(*=======================================================*)
	1:	(* Warte auf Kommando *)
		IF st_ecd_cmd.enu_cmd > NO_COMMAND THEN
			IF st_ecd_cmd.enu_cmd <= HALT_AXIS THEN
				(* Wichtige Kommandos werden mit Direktsprung ausgeführt, um Zykluszeit zu sparen *)
				IF st_ecd_cmd.enu_cmd = HALT_AXIS THEN
					fb_state_entry.i16_next_step := 120;
				ELSIF st_ecd_cmd.enu_cmd = STOP_AXIS THEN
					fb_state_entry.i16_next_step := 130;
				ELSE
					fb_state_entry.i16_next_step := 10;	(* Motionbefehle *)
				END_IF
			ELSE
				fb_state_entry.i16_next_step := 500;	(* Parameter für Achsen *)
			END_IF
		END_IF

(*=======================Motionbefehle================================*)
	10:	(* Power OFF NC-Achse *)
		fb_ton_cmd_timeout.IN := TRUE;
		IF st_ecd_cmd.enu_cmd = POWER_DISABLE THEN
			mc_power_axis.Enable := FALSE;
			fb_state_entry.i16_next_step := 11;
		ELSE
			fb_ton_cmd_timeout.IN := FALSE;
			fb_state_entry.i16_next_step := 20;
		END_IF
	11:
		CASE i16_achstyp OF
			LINEAR, RUND:
				IF NOT mc_power_axis.Status AND NOT st_masterachse.Status.Operational THEN
					fb_state_entry.i16_next_step := 999;
				ELSIF NOT mc_power_axis.Busy AND mc_power_axis.Error THEN
					err_id := mc_power_axis.ErrorID;
					st_ecd_cmd.meldungen.sm_power_disable := TRUE;
					fb_state_entry.i16_next_step := 1000;
				END_IF
			LINEAR_VIRTUELL, RUND_VIRTUELL:
				IF NOT mc_power_axis.Busy AND mc_power_axis.Error THEN
					err_id := mc_power_axis.ErrorID;
					st_ecd_cmd.meldungen.sm_power_disable := TRUE;
					fb_state_entry.i16_next_step := 1000;
				ELSE
					fb_state_entry.i16_next_step := 999;
				END_IF
			SERVOKLEMME7201:
				IF NOT mc_power_axis.Status AND NOT st_masterachse.Status.Operational THEN
					fb_state_entry.i16_next_step := 999;
				ELSIF NOT mc_power_axis.Busy AND mc_power_axis.Error THEN
					err_id := mc_power_axis.ErrorID;
					st_ecd_cmd.meldungen.sm_power_disable := TRUE;
					fb_state_entry.i16_next_step := 1000;
				END_IF
		END_CASE

(*=======================================================*)
	20:	(* Reset NC-Achse und Servokontroller*)
		IF	st_ecd_cmd.enu_cmd = RESET OR
			st_masterachse.Status.DriveDeviceError OR
			st_masterachse.Status.Error
			 THEN
			fb_state_entry.i16_next_step := 21;
		ELSE
			fb_state_entry.i16_next_step := 30;
		END_IF
	21:	(*  Reset AX5000 Fehler  *)
		CASE i16_achstyp OF
			LINEAR, RUND:
				IF NOT st_masterachse.Status.DriveDeviceError THEN
					fb_state_entry.i16_next_step := 24;
				ELSE
					fb_ton_cmd_timeout.IN := TRUE;
					fb_soe_reset.Execute := TRUE;
					IF fb_soe_reset.Busy THEN
						fb_state_entry.i16_next_step := 22;
					END_IF
				END_IF
			LINEAR_VIRTUELL, RUND_VIRTUELL, SERVOKLEMME7201:
				fb_state_entry.i16_next_step := 24;
		END_CASE
	22:
		IF NOT fb_soe_reset.Busy THEN
			IF  fb_soe_reset.Error THEN
				st_ecd_cmd.meldungen.sm_reset := TRUE;
				fb_state_entry.i16_next_step := 1000;
			ELSE
				fb_soe_reset.Execute := FALSE;
				fb_state_entry.i16_next_step := 23;
			END_IF
		END_IF
	23:
		IF NOT st_masterachse.Status.DriveDeviceError THEN
			fb_ton_cmd_timeout.IN := FALSE;
			fb_state_entry.i16_next_step := 24;
		END_IF
	24:	(* Reset NC-Achsfehler *)
		CASE i16_achstyp OF
			LINEAR, RUND, LINEAR_VIRTUELL, RUND_VIRTUELL:
				IF NOT st_masterachse.Status.Error THEN
					fb_state_entry.i16_next_step := 26;
				ELSE
					fb_ton_cmd_timeout.IN := TRUE;
					mc_reset_axis.Execute := TRUE;
					IF mc_reset_axis.Busy THEN
						fb_state_entry.i16_next_step := 25;
					END_IF
				END_IF
			SERVOKLEMME7201:
				IF NOT st_masterachse.Status.Error AND NOT st_masterachse.Status.DriveDeviceError THEN
					fb_state_entry.i16_next_step := 26;
				ELSE
					fb_ton_cmd_timeout.IN := TRUE;
					mc_reset_axis.Execute := TRUE;
					IF mc_reset_axis.Busy THEN
						fb_state_entry.i16_next_step := 25;
					END_IF
				END_IF
		END_CASE
	25:
		IF NOT st_masterachse.Status.Error THEN
			mc_reset_axis.Execute := FALSE;
			fb_ton_cmd_timeout.IN := FALSE;
			fb_state_entry.i16_next_step := 26;
		END_IF
	26:
		IF st_ecd_cmd.enu_cmd = RESET THEN
			fb_state_entry.i16_next_step := 999;
		ELSE
			fb_state_entry.i16_next_step := 30;
		END_IF

(*=======================================================*)
	30:	(* Power ON NC-Achse *)
		CASE i16_achstyp OF
			LINEAR, RUND:
				fb_ton_cmd_timeout.IN := TRUE;
				IF	(st_ecd_cmd.enu_cmd > POWER_DISABLE AND st_ecd_cmd.enu_cmd < HALT_AXIS)  AND
					(NOT st_masterachse.Status.Operational OR
					(st_ecd_cmd.enu_cmd = POWER_ENABLE AND NOT st_masterachse.Status.Operational))
					THEN
						fb_state_entry.i16_next_step := 31;
				ELSE
					fb_ton_cmd_timeout.IN := FALSE;
					fb_state_entry.i16_next_step := 40;
				END_IF
			LINEAR_VIRTUELL, RUND_VIRTUELL, SERVOKLEMME7201:
				IF	st_ecd_cmd.enu_cmd > POWER_DISABLE AND st_ecd_cmd.enu_cmd < HALT_AXIS AND
					NOT mc_power_axis.Status
					THEN
						fb_state_entry.i16_next_step := 31;
				ELSE
					fb_ton_cmd_timeout.IN := FALSE;
					fb_state_entry.i16_next_step := 40;
				END_IF
		END_CASE
	31:
		mc_power_axis.Enable_Positive := TRUE;
		mc_power_axis.Enable_Negative := TRUE;
		mc_power_axis.Enable := TRUE;
		IF mc_power_axis.Busy THEN
			fb_ton_vz.PT := t#1s;
			fb_ton_vz.IN := TRUE;
			fb_state_entry.i16_next_step := 32;
		END_IF
	32:
		IF mc_power_axis.Status AND st_masterachse.Status.Operational  THEN
			IF st_ecd_cmd.enu_cmd = POWER_ENABLE THEN
				fb_state_entry.i16_next_step := 999;
			ELSE
				fb_ton_cmd_timeout.IN := FALSE;
				fb_state_entry.i16_next_step := 40;
			END_IF
		ELSIF mc_power_axis.Error AND fb_ton_vz.Q THEN
			st_ecd_cmd.meldungen.sm_power_enable := TRUE;
			err_id := mc_power_axis.ErrorID;
			fb_state_entry.i16_next_step := 1000;
		END_IF
		IF st_ecd_cmd.enu_cmd = HALT_AXIS THEN
			fb_ton_cmd_timeout.IN := FALSE;
			fb_ton_vz.IN := FALSE;
			fb_state_entry.i16_next_step := 121;
		END_IF
		IF st_ecd_cmd.enu_cmd = STOP_AXIS THEN
			fb_ton_cmd_timeout.IN := FALSE;
			fb_ton_vz.IN := FALSE;
			fb_state_entry.i16_next_step := 131;
		END_IF

(*=======================================================*)
	40:	(* Abfrage Referenzieren und Ref-Art *)
		IF st_ecd_cmd.enu_cmd = HOME THEN
			IF b_refsensor_vorhanden THEN
				mc_referenzmodus := MC_DefaultHoming;
			ELSE
				mc_referenzmodus := MC_Direct;
			END_IF
			st_position.r_referenz := 0.0;
			fb_state_entry.i16_next_step := 41;
		ELSE
			fb_ton_cmd_timeout.IN := FALSE;
			fb_state_entry.i16_next_step := 50;
		END_IF
	41:	(* Start Homing *)
		mc_home_axis.Execute := TRUE;
		mc_home_axis.Options.ClearPositionLag := TRUE;
		IF mc_home_axis.Busy THEN
			fb_state_entry.i16_next_step := 42;
		END_IF
	42:
		IF mc_home_axis.Done THEN
			mc_home_axis.Execute := FALSE;
			fb_state_entry.i16_next_step := 999;
		END_IF
		IF NOT mc_home_axis.Busy AND mc_home_axis.Error THEN
			st_ecd_cmd.meldungen.sm_home := TRUE;
			err_id := mc_home_axis.ErrorID;
			fb_state_entry.i16_next_step := 1000;
		END_IF
		IF st_ecd_cmd.enu_cmd = HALT_AXIS THEN
			mc_home_axis.Execute := FALSE;
			fb_ton_cmd_timeout.IN := FALSE;
			fb_state_entry.i16_next_step := 121;
		END_IF
		IF st_ecd_cmd.enu_cmd = STOP_AXIS THEN
			mc_home_axis.Execute := FALSE;
			fb_ton_cmd_timeout.IN := FALSE;
			fb_state_entry.i16_next_step := 131;
		END_IF

(*=======================================================*)
	50:	(* Jog vorwärts *)
		IF st_ecd_cmd.enu_cmd = JOG_VORWAERTS THEN
			fb_state_entry.i16_next_step := 51;
		ELSE
			fb_state_entry.i16_next_step := 55;
		END_IF
	51:
		b_jog_vorwaerts_execute := TRUE;
		IF mc_jog_axis.Active THEN
			fb_state_entry.i16_next_step := 52;
		ELSIF mc_jog_axis.Error THEN
			st_ecd_cmd.meldungen.sm_jog_vorwaerts := TRUE;
			fb_state_entry.i16_next_step := FEHLER;
		END_IF
	52:
		IF st_ecd_cmd.enu_cmd = JOG_STOP OR st_ecd_cmd.enu_cmd = JOG_RUECKWAERTS THEN
			fb_state_entry.i16_next_step := 61;
		END_IF

		IF st_ecd_cmd.enu_cmd = HALT_AXIS THEN
			mc_movemodulo_axis.Execute := FALSE;
			fb_ton_cmd_timeout.IN := FALSE;
			fb_state_entry.i16_next_step := 121;
		END_IF
		IF st_ecd_cmd.enu_cmd = STOP_AXIS THEN
			mc_movemodulo_axis.Execute := FALSE;
			fb_ton_cmd_timeout.IN := FALSE;
			fb_state_entry.i16_next_step := 131;
		END_IF

(*=======================================================*)
	55:	(* Jog rückwärts *)
		IF st_ecd_cmd.enu_cmd = JOG_RUECKWAERTS THEN
			fb_state_entry.i16_next_step := 56;
		ELSE
			fb_state_entry.i16_next_step := 60;
		END_IF

	56:
		b_jog_rueckwaerts_execute := TRUE;
		IF mc_jog_axis.Active THEN
			fb_state_entry.i16_next_step := 57;
		ELSIF mc_jog_axis.Error THEN
			st_ecd_cmd.meldungen.sm_jog_rueckwaerts := TRUE;
			fb_state_entry.i16_next_step := FEHLER;
		END_IF
	57:
		IF st_ecd_cmd.enu_cmd = JOG_STOP OR st_ecd_cmd.enu_cmd = JOG_VORWAERTS THEN
			fb_state_entry.i16_next_step := 61;
		END_IF

		IF st_ecd_cmd.enu_cmd = HALT_AXIS THEN
			mc_movemodulo_axis.Execute := FALSE;
			fb_ton_cmd_timeout.IN := FALSE;
			fb_state_entry.i16_next_step := 121;
		END_IF
		IF st_ecd_cmd.enu_cmd = STOP_AXIS THEN
			mc_movemodulo_axis.Execute := FALSE;
			fb_ton_cmd_timeout.IN := FALSE;
			fb_state_entry.i16_next_step := 131;
		END_IF

(*=======================================================*)
	60:	(* Jog Stop *)
		IF st_ecd_cmd.enu_cmd = JOG_STOP THEN
			fb_state_entry.i16_next_step := 61;
		ELSE
			fb_state_entry.i16_next_step := 70;
		END_IF
	61:
		b_jog_vorwaerts_execute := FALSE;
		b_jog_rueckwaerts_execute := FALSE;
		fb_state_entry.i16_next_step := 999;

(*=======================================================*)
	70:	(* Move absolute *)
		IF st_ecd_cmd.enu_cmd = MOVE_ABSOLUTE THEN
			fb_state_entry.i16_next_step := 71;
		ELSE
			fb_state_entry.i16_next_step := 80;
		END_IF
	71:
		IF ABS(st_masterachse.NcToPlc.ActPos -  st_position.r_soll ) < 0.05 THEN
			fb_state_entry.i16_next_step := 999;
		ELSE
			mc_moveabsolute_axis.Execute := TRUE;
		END_IF
		IF mc_moveabsolute_axis.Busy THEN
			fb_state_entry.i16_next_step := 72;
		END_IF
	72:
		IF mc_moveabsolute_axis.Done THEN
			mc_moveabsolute_axis.Execute := FALSE;
			fb_state_entry.i16_next_step := 999;
		END_IF
		IF NOT mc_moveabsolute_axis.Busy AND mc_moveabsolute_axis.Error THEN
			st_ecd_cmd.meldungen.sm_move_absolute := TRUE;
			err_id := mc_moveabsolute_axis.ErrorID;
			fb_state_entry.i16_next_step := 1000;
		END_IF
		IF st_ecd_cmd.enu_cmd = HALT_AXIS THEN
			mc_moveabsolute_axis.Execute := FALSE;
			fb_ton_cmd_timeout.IN := FALSE;
			fb_state_entry.i16_next_step := 121;
		END_IF
		IF st_ecd_cmd.enu_cmd = STOP_AXIS THEN
			mc_moveabsolute_axis.Execute := FALSE;
			fb_ton_cmd_timeout.IN := FALSE;
			fb_state_entry.i16_next_step := 131;
		END_IF

		(* Move-Kommando für folgende Bewegung *)
		IF st_ecd_cmd.enu_cmd = MOVE_ABSOLUTE_NEXT THEN
			fb_state_entry.i16_next_step := 74;
		END_IF
	74:
		IF ABS(st_masterachse.NcToPlc.ActPos -  st_position.r_soll ) < 0.05 THEN
			fb_state_entry.i16_next_step := 999;
		ELSE
			mc_moveabsolutenext_axis.Execute := TRUE;
		END_IF
		IF mc_moveabsolutenext_axis.Busy THEN
			fb_state_entry.i16_next_step := 75;
		END_IF
	75:
		IF mc_moveabsolutenext_axis.Done THEN
			mc_moveabsolute_axis.Execute := FALSE;
			mc_moveabsolutenext_axis.Execute := FALSE;
			fb_state_entry.i16_next_step := 999;
		END_IF
		IF NOT mc_moveabsolutenext_axis.Busy AND mc_moveabsolutenext_axis.Error THEN
			st_ecd_cmd.meldungen.sm_move_absolute := TRUE;
			err_id := mc_moveabsolutenext_axis.ErrorID;
			fb_state_entry.i16_next_step := 1000;
		END_IF
		IF st_ecd_cmd.enu_cmd = HALT_AXIS THEN
			mc_moveabsolute_axis.Execute := FALSE;
			mc_moveabsolutenext_axis.Execute := FALSE;
			fb_ton_cmd_timeout.IN := FALSE;
			fb_state_entry.i16_next_step := 121;
		END_IF
		IF st_ecd_cmd.enu_cmd = STOP_AXIS THEN
			mc_moveabsolute_axis.Execute := FALSE;
			mc_moveabsolutenext_axis.Execute := FALSE;
			fb_ton_cmd_timeout.IN := FALSE;
			fb_state_entry.i16_next_step := 131;
		END_IF

(*=======================================================*)
	80:	(* Move relative *)
		IF st_ecd_cmd.enu_cmd = MOVE_RELATIVE THEN
			fb_state_entry.i16_next_step := 81;
		ELSE
			fb_state_entry.i16_next_step := 90;
		END_IF
	81:
		mc_moverelative_axis.Execute := TRUE;
		IF mc_moverelative_axis.Busy THEN
			fb_state_entry.i16_next_step := 82;
		END_IF
	82:
		IF mc_moverelative_axis.Done THEN
			mc_moverelative_axis.Execute := FALSE;
			fb_state_entry.i16_next_step := 999;
		END_IF
		IF NOT mc_moverelative_axis.Busy AND mc_moverelative_axis.Error THEN
			st_ecd_cmd.meldungen.sm_move_relative := TRUE;
			err_id := mc_moverelative_axis.ErrorID;
			fb_state_entry.i16_next_step := 1000;
		END_IF
		IF st_ecd_cmd.enu_cmd = HALT_AXIS THEN
			mc_moverelative_axis.Execute := FALSE;
			fb_ton_cmd_timeout.IN := FALSE;
			fb_state_entry.i16_next_step := 121;
		END_IF
		IF st_ecd_cmd.enu_cmd = STOP_AXIS THEN
			mc_moverelative_axis.Execute := FALSE;
			fb_ton_cmd_timeout.IN := FALSE;
			fb_state_entry.i16_next_step := 131;
		END_IF

(*=======================================================*)
	90:	(* Move velocity *)
		IF st_ecd_cmd.enu_cmd = MOVE_VELOCITY THEN
			fb_state_entry.i16_next_step := 91;
		ELSE
			fb_state_entry.i16_next_step := 100;
		END_IF
	91:
		mc_movevelocity_axis.Execute := TRUE;
		IF mc_movevelocity_axis.Busy THEN
			fb_state_entry.i16_next_step := 92;
		END_IF
	92:
		IF mc_movevelocity_axis.InVelocity THEN
			mc_movevelocity_axis.Execute := FALSE;
			fb_state_entry.i16_next_step := 999;
		END_IF
		IF NOT mc_movevelocity_axis.Busy AND mc_movevelocity_axis.Error THEN
			st_ecd_cmd.meldungen.sm_move_velocity := TRUE;
			err_id := mc_movevelocity_axis.ErrorID;
			fb_state_entry.i16_next_step := 1000;
		END_IF
		IF st_ecd_cmd.enu_cmd = HALT_AXIS THEN
			mc_movevelocity_axis.Execute := FALSE;
			fb_ton_cmd_timeout.IN := FALSE;
			fb_state_entry.i16_next_step := 121;
		END_IF
		IF st_ecd_cmd.enu_cmd = STOP_AXIS THEN
			mc_movevelocity_axis.Execute := FALSE;
			fb_ton_cmd_timeout.IN := FALSE;
			fb_state_entry.i16_next_step := 131;
		END_IF

(*=======================================================*)
	100:	(* Move modulo *)
		IF st_ecd_cmd.enu_cmd = MOVE_MODULO THEN
			fb_state_entry.i16_next_step := 101;
		ELSE
			fb_state_entry.i16_next_step := 103;
		END_IF
	101:
		IF ABS(st_masterachse.NcToPlc.ModuloActPos -  st_position.r_soll ) < 0.3 THEN
			fb_state_entry.i16_next_step := 999;
		ELSE
			mc_movemodulo_axis.Execute := TRUE;
		END_IF
		IF mc_movemodulo_axis.Busy THEN
			fb_state_entry.i16_next_step := 102;
		END_IF
	102:
		IF mc_movemodulo_axis.Done THEN
			mc_movemodulo_axis.Execute := FALSE;
			fb_state_entry.i16_next_step := 999;
		END_IF

		IF NOT mc_movemodulo_axis.Busy AND mc_movemodulo_axis.Error THEN
			st_ecd_cmd.meldungen.sm_move_modulo := TRUE;
			err_id := mc_movemodulo_axis.ErrorID;
			fb_state_entry.i16_next_step := 1000;
		END_IF
		IF st_ecd_cmd.enu_cmd = HALT_AXIS THEN
			mc_movemodulo_axis.Execute := FALSE;
			fb_ton_cmd_timeout.IN := FALSE;
			fb_state_entry.i16_next_step := 121;
		END_IF
		IF st_ecd_cmd.enu_cmd = STOP_AXIS THEN
			mc_movemodulo_axis.Execute := FALSE;
			fb_ton_cmd_timeout.IN := FALSE;
			fb_state_entry.i16_next_step := 131;
		END_IF

(*=======================================================*)
	103:
		(*Touch Probe checken*)
		IF	fb_state_entry.E THEN
			mc_abort_trigger.Execute:=TRUE;
		END_IF

		IF st_ecd_cmd.enu_cmd = MOVE_TOUCH_PROBE THEN

			(*Touch Probe darf nicht betätigt sein*)
			IF	(b_FallingEdge AND NOT b_TriggerInput) OR
				(NOT b_FallingEdge AND b_TriggerInput)  THEN
				st_ecd_cmd.meldungen.sm_touch_probe_defect := TRUE;		(*Messtaster defekt*)
				fb_state_entry.i16_next_step := FEHLER;

			ELSIF mc_abort_trigger.Done THEN
				lr_RecPos:=0;
				fb_state_entry.i16_next_step := 104;
			END_IF

		ELSE
			fb_state_entry.i16_next_step := 110;
		END_IF

		IF	fb_state_entry.X THEN
			mc_abort_trigger.Execute:=FALSE;
		END_IF

	104:
		(* Move absolute (Position muss hinter dem Touch Probe liegen => der Restweg wird gelöscht)*)
		IF 	ABS(st_masterachse.NcToPlc.ActPos -  st_position.r_soll ) < 0.05 THEN
			fb_state_entry.i16_next_step := 999;
		ELSE
			mc_moveabsolute_axis.Execute := TRUE;
			mc_touch_probe.Execute:=TRUE;
		END_IF
		IF 	mc_moveabsolute_axis.Busy THEN
			fb_state_entry.i16_next_step := 105;
		END_IF

	105:
		(*Achsposition wurde erreicht ohne Taster Event*)
		IF 	mc_moveabsolute_axis.Done THEN
			fb_state_entry.i16_next_step := 999;
		END_IF

		(*Achse anhalten wenn Touch Probe betätigt wird*)
		IF 	mc_moveabsolute_axis.Busy AND
			(b_TriggerInput = NOT b_FallingEdge OR
			mc_touch_probe.Done) THEN
			fb_state_entry.i16_next_step := 131;
		END_IF

		(*Übergabe Rec Position*)
		IF	mc_touch_probe.Done THEN
			lr_RecPos:=mc_touch_probe.RecordedPosition;
		END_IF

		(*Fehler Achse*)
		IF 	NOT mc_moveabsolute_axis.Busy AND mc_moveabsolute_axis.Error THEN
			st_ecd_cmd.meldungen.sm_move_absolute := TRUE;
			err_id := mc_moveabsolute_axis.ErrorID;
			fb_state_entry.i16_next_step := FEHLER;
		END_IF

		(*Fehler Touch Probe*)
		IF  	mc_touch_probe.Error THEN
			st_ecd_cmd.meldungen.sm_touch_probe_err := TRUE;
			err_id := mc_touch_probe.ErrorID;
			fb_state_entry.i16_next_step := FEHLER;
		END_IF

		IF	fb_state_entry.X THEN
			fb_ton_cmd_timeout.IN := FALSE;
			mc_moveabsolute_axis.Execute := FALSE;
			mc_touch_probe.Execute:=FALSE;
		END_IF

(*=======================================================*)
	110:	(* Position *)
		IF st_ecd_cmd.enu_cmd = SET_POSITION THEN
			fb_state_entry.i16_next_step := 111;
		ELSE
			fb_state_entry.i16_next_step := 121;
		END_IF
	111:
		(* Soll- und Istposition werden auf den gleichen Wert gesetzt und somit der Schleppfehler gelöscht. *)
		mc_setposition_axis.Options.ClearPositionLag := TRUE;
		mc_setposition_axis.Options.EncoderIndex := 0;
		mc_setposition_axis.Options.SelectEncoderIndex := FALSE;
		mc_setposition_axis.Execute := TRUE;
		IF mc_setposition_axis.Busy THEN
			fb_state_entry.i16_next_step := 112;
		END_IF
	112:
		IF mc_setposition_axis.Done THEN
			mc_setposition_axis.Execute := FALSE;
			fb_state_entry.i16_next_step := 999;
		END_IF
		IF NOT mc_setposition_axis.Busy AND mc_setposition_axis.Error THEN
			st_ecd_cmd.meldungen.sm_setposition := TRUE;
			err_id := mc_setposition_axis.ErrorID;
			fb_state_entry.i16_next_step := 1000;
		END_IF
		IF st_ecd_cmd.enu_cmd = HALT_AXIS THEN
			mc_setposition_axis.Execute := FALSE;
			fb_ton_cmd_timeout.IN := FALSE;
			fb_state_entry.i16_next_step := 121;
		END_IF
		IF st_ecd_cmd.enu_cmd = STOP_AXIS THEN
			mc_setposition_axis.Execute := FALSE;
			fb_ton_cmd_timeout.IN := FALSE;
			fb_state_entry.i16_next_step := 131;
		END_IF

(*=======================================================*)
	120:	(* Halt *)
		fb_ton_cmd_timeout.IN := TRUE;
		IF st_ecd_cmd.enu_cmd = HALT_AXIS THEN
			fb_state_entry.i16_next_step := 121;
		ELSE
			fb_ton_cmd_timeout.IN := FALSE;
			fb_state_entry.i16_next_step := 131;
		END_IF
	121:
		mc_halt_axis.Execute := TRUE;
		IF mc_halt_axis.Busy THEN
			fb_state_entry.i16_next_step := 122;
		END_IF
	122:
		IF mc_halt_axis.Done THEN
			mc_halt_axis.Execute := FALSE;
			fb_state_entry.i16_next_step := 123;
		END_IF
		IF NOT mc_halt_axis.Busy AND mc_halt_axis.Error THEN
			st_ecd_cmd.meldungen.sm_halt_axis := TRUE;
			err_id := mc_halt_axis.ErrorID;
			fb_state_entry.i16_next_step := 1000;
		END_IF
	123:
		IF	NOT st_masterachse.Status.ConstantVelocity AND
			NOT st_masterachse.Status.Accelerating AND
			NOT st_masterachse.Status.Decelerating
			THEN
				fb_state_entry.i16_next_step := 999;
		END_IF

(*=======================================================*)
	130: (* Stop *)
		fb_ton_cmd_timeout.IN := TRUE;
		IF st_ecd_cmd.enu_cmd = STOP_AXIS THEN
			fb_state_entry.i16_next_step := 131;
		ELSE
			fb_ton_cmd_timeout.IN := FALSE;
			fb_state_entry.i16_next_step := 140;
		END_IF
	131:
		mc_stop_axis.Execute := TRUE;
		IF mc_stop_axis.Busy THEN
			fb_state_entry.i16_next_step := 132;
		END_IF
	132:
		IF mc_stop_axis.Done THEN
			mc_stop_axis.Execute := FALSE;
			fb_state_entry.i16_next_step := 133;
		END_IF
		IF mc_stop_axis.Error THEN
			st_ecd_cmd.meldungen.sm_stop_axis := TRUE;
			err_id := mc_stop_axis.ErrorID;
			fb_state_entry.i16_next_step := 1000;
		END_IF
	133:
		IF 	NOT st_masterachse.Status.ConstantVelocity AND
			NOT st_masterachse.Status.Accelerating AND
			NOT st_masterachse.Status.Decelerating
			THEN
				fb_state_entry.i16_next_step := 999;
		END_IF

(*=======================================================*)
	140:	(* Frei *)
		fb_state_entry.i16_next_step := 500;

(*======================Parameterbefehle=================================*)
	500:	(* Schreibe einen Parameter an den Antrieb *)
		fb_ton_cmd_timeout.IN := TRUE;
		IF st_ecd_cmd.enu_cmd = SOE_WRITE_PARAM THEN
			fb_state_entry.i16_next_step := 501;
		ELSE
			fb_ton_cmd_timeout.IN := FALSE;
			fb_state_entry.i16_next_step := 510;
		END_IF
	501:
		fb_soe_write.Execute := TRUE;
		IF fb_soe_write.Busy THEN
			fb_state_entry.i16_next_step := 502;
		END_IF
	502:
		IF NOT fb_soe_write.Busy THEN
			fb_soe_write.Execute := FALSE;
			IF fb_soe_write.Error THEN
				st_ecd_cmd.meldungen.sm_write_soe_parameter := TRUE;
				fb_state_entry.i16_next_step := 1000;
			ELSE
				fb_state_entry.i16_next_step := 999;
			END_IF
		END_IF

(*=======================================================*)
	510:	(* Lesen eines Parameter vom Antrieb *)
		fb_ton_cmd_timeout.IN := TRUE;
		IF st_ecd_cmd.enu_cmd = SOE_READ_PARAM THEN
			fb_state_entry.i16_next_step := 511;
		ELSE
			fb_ton_cmd_timeout.IN := FALSE;
			fb_state_entry.i16_next_step := 520;
		END_IF
	511:
		fb_soe_read.Execute := TRUE;
		IF fb_soe_read.Busy THEN
			fb_state_entry.i16_next_step := 512;
		END_IF
	512:
		IF NOT fb_soe_read.Busy THEN
			fb_soe_write.Execute := FALSE;
			IF fb_soe_read.Error THEN
				st_ecd_cmd.meldungen.sm_read_soe_parameter := TRUE;
				fb_state_entry.i16_next_step := 1000;
			ELSE
				fb_state_entry.i16_next_step := 999;
			END_IF
		END_IF

(*=======================================================*)
	520:	(* Schreibe einen Parameter an die NC-Achse *)
		fb_ton_cmd_timeout.IN := TRUE;
		IF st_ecd_cmd.enu_cmd = WRITE_NC_PARAMETER THEN
			fb_state_entry.i16_next_step := 521;
		ELSE
			fb_ton_cmd_timeout.IN := FALSE;
			fb_state_entry.i16_next_step := 530;
		END_IF
	521:
		mc_write_nc_parameter.Execute := TRUE;
		IF mc_write_nc_parameter.Busy THEN
			fb_state_entry.i16_next_step := 522;
		END_IF
	522:
		IF NOT mc_write_nc_parameter.Busy THEN
			mc_write_nc_parameter.Execute := FALSE;
			IF mc_write_nc_parameter.Error THEN
				st_ecd_cmd.meldungen.sm_write_nc_parameter := TRUE;
				fb_state_entry.i16_next_step := 1000;
			ELSE
				fb_state_entry.i16_next_step := 999;
			END_IF
		END_IF

(*=======================================================*)
	530:	(* Lesen eines Parameter vom der NC-Achse *)
		fb_ton_cmd_timeout.IN := TRUE;
		IF st_ecd_cmd.enu_cmd = READ_NC_PARAMETER THEN
			fb_state_entry.i16_next_step := 531;
		ELSE
			fb_ton_cmd_timeout.IN := FALSE;
			fb_state_entry.i16_next_step := 540;
		END_IF
	531:
		mc_read_nc_parameter.Enable := TRUE;
		IF mc_read_nc_parameter.Busy THEN
			fb_state_entry.i16_next_step := 532;
		END_IF
	532:
		IF NOT mc_read_nc_parameter.Busy THEN
			mc_read_nc_parameter.Enable := FALSE;
			IF mc_read_nc_parameter.Error THEN
				st_ecd_cmd.meldungen.sm_read_nc_parameter := TRUE;
				fb_state_entry.i16_next_step := 1000;
			ELSE
				fb_state_entry.i16_next_step := 999;
			END_IF
		END_IF

(*=======================================================*)
	540:	(* Schreibe einen beliebigen ADS-Parameter an die NC-Achse *)
		fb_ton_cmd_timeout.IN := TRUE;
		IF st_ecd_cmd.enu_cmd = WRITE_ADS_PARAMETER THEN
			fb_state_entry.i16_next_step := 541;
		ELSE
			fb_ton_cmd_timeout.IN := FALSE;
			fb_state_entry.i16_next_step := 550;
		END_IF
	541:
		fb_ads_write.WRITE := TRUE;
		IF fb_ads_write.BUSY THEN
			fb_state_entry.i16_next_step := 542;
		END_IF
	542:
		IF NOT fb_ads_write.BUSY THEN
			fb_ads_write.WRITE := FALSE;
			IF fb_ads_write.ERR THEN
				st_ecd_cmd.meldungen.sm_write_ads_parameter := TRUE;
				fb_state_entry.i16_next_step := 1000;
			ELSE
				fb_state_entry.i16_next_step := 999;
			END_IF
		END_IF

(*=======================================================*)
	550:	(* Lesen einen beliebigenADS-Parameter vom der NC-Achse *)
		fb_ton_cmd_timeout.IN := TRUE;
		IF st_ecd_cmd.enu_cmd = READ_ADS_PARAMETER THEN
			fb_state_entry.i16_next_step := 551;
		ELSE
			fb_ton_cmd_timeout.IN := FALSE;
			fb_state_entry.i16_next_step := 560;
		END_IF
	551:
		fb_ads_read.READ := TRUE;
		IF fb_ads_read.BUSY THEN
			fb_state_entry.i16_next_step := 552;
		END_IF
	552:
		IF NOT fb_ads_read.BUSY THEN
			fb_ads_read.READ := FALSE;
			IF fb_ads_read.ERR THEN
				st_ecd_cmd.meldungen.sm_read_ads_parameter := TRUE;
				fb_state_entry.i16_next_step := 1000;
			ELSE
				fb_state_entry.i16_next_step := 999;
			END_IF
		END_IF

(*=======================================================*)
	560:	(* Schreibe die neuen EcSoe Parameter an den Antrieb *)
		fb_ton_cmd_timeout.IN := TRUE;
		IF st_ecd_cmd.enu_cmd = ECCOESDO_WRITE_PARAM THEN
			fb_state_entry.i16_next_step := 561;
		ELSE
			fb_ton_cmd_timeout.IN := FALSE;
			fb_state_entry.i16_next_step := 570;
		END_IF
	561:
		fb_ec_coe_sdo_write_ex.bExecute := TRUE;
		IF fb_ec_coe_sdo_write_ex.bBusy THEN
			fb_state_entry.i16_next_step := 562;
		END_IF
	562:
		IF NOT fb_ec_coe_sdo_write_ex.bBusy THEN
			fb_ec_coe_sdo_write_ex.bExecute := FALSE;
			IF fb_ec_coe_sdo_write_ex.bError THEN
				st_ecd_cmd.meldungen.sm_ec_coe_sdo_write_ex := TRUE;
				fb_state_entry.i16_next_step := 1000;
			ELSE
				fb_state_entry.i16_next_step := 999;
			END_IF
		END_IF

(*=======================================================*)
	570:	(* Lese die neuen EcSoe Parameter an den Antrieb *)
		fb_ton_cmd_timeout.IN := TRUE;
		IF st_ecd_cmd.enu_cmd = ECCOESDO_READ_PARAM THEN
			fb_state_entry.i16_next_step := 571;
		ELSE
			fb_ton_cmd_timeout.IN := FALSE;
			fb_state_entry.i16_next_step := 580;
		END_IF
	571:
		fb_ec_coe_sdo_read_ex.bExecute := TRUE;
		IF fb_ec_coe_sdo_read_ex.bBusy THEN
			fb_state_entry.i16_next_step := 572;
		END_IF
	572:
		IF NOT fb_ec_coe_sdo_read_ex.bBusy THEN
			fb_ec_coe_sdo_read_ex.bExecute := FALSE;
			IF fb_ec_coe_sdo_read_ex.bError THEN
				st_ecd_cmd.meldungen.sm_ec_coe_sdo_read_ex := TRUE;
				fb_state_entry.i16_next_step := 1000;
			ELSE
				fb_state_entry.i16_next_step := 999;
			END_IF
		END_IF

(*=======================================================*)
	580:	(* Frei *)
		fb_state_entry.i16_next_step := 999;

(*=======================================================*)
	999:	(* Ende - Befehl wurde korrekt abgearbeitet *)
		st_ecd_cmd.enu_cmd := NO_COMMAND;
		fb_ton_cmd_timeout.IN := FALSE;
		fb_ton_vz.IN := FALSE;

		b_jog_vorwaerts_execute := FALSE;
		b_jog_rueckwaerts_execute := FALSE;

		mc_reset_axis.Execute := FALSE;
		mc_home_axis.Execute := FALSE;
		mc_moveabsolute_axis.Execute := FALSE;
		mc_moverelative_axis.Execute := FALSE;
		mc_movevelocity_axis.Execute := FALSE;
		mc_movemodulo_axis.Execute := FALSE;
		mc_setposition_axis.Execute := FALSE;
		mc_halt_axis.Execute := FALSE;
		mc_stop_axis.Execute := FALSE;
		fb_soe_reset.Execute := FALSE;
		fb_soe_write.Execute := FALSE;
		fb_soe_read.Execute := FALSE;
		mc_write_nc_parameter.Execute := FALSE;
		mc_read_nc_parameter.Enable := FALSE;
		fb_ads_write.WRITE := FALSE;
		fb_ads_read.READ := FALSE;
		fb_ec_coe_sdo_write_ex.bExecute := FALSE;
		fb_ec_coe_sdo_read_ex.bExecute := FALSE;

		st_ecd_cmd.meldungen.sm_power_enable := FALSE;
		st_ecd_cmd.meldungen.sm_power_disable := FALSE;
		st_ecd_cmd.meldungen.sm_reset := FALSE;
		st_ecd_cmd.meldungen.sm_home := FALSE;
		st_ecd_cmd.meldungen.sm_setposition := FALSE;
		st_ecd_cmd.meldungen.sm_jog_vorwaerts := FALSE;
		st_ecd_cmd.meldungen.sm_jog_rueckwaerts := FALSE;
		st_ecd_cmd.meldungen.sm_move_absolute := FALSE;
		st_ecd_cmd.meldungen.sm_move_relative := FALSE;
		st_ecd_cmd.meldungen.sm_move_velocity := FALSE;
		st_ecd_cmd.meldungen.sm_move_modulo := FALSE;
		st_ecd_cmd.meldungen.sm_stop_axis := FALSE;
		st_ecd_cmd.meldungen.sm_halt_axis := FALSE;
		st_ecd_cmd.meldungen.sm_motion_command_timeout := FALSE;
		st_ecd_cmd.meldungen.sm_limit_positiv_erreicht := FALSE;
		st_ecd_cmd.meldungen.sm_limit_negativ_erreicht := FALSE;
		st_ecd_cmd.meldungen.sm_write_soe_parameter := FALSE;
		st_ecd_cmd.meldungen.sm_read_soe_parameter := FALSE;
		st_ecd_cmd.meldungen.sm_write_nc_parameter := FALSE;
		st_ecd_cmd.meldungen.sm_read_nc_parameter := FALSE;
		st_ecd_cmd.meldungen.sm_write_ads_parameter := FALSE;
		st_ecd_cmd.meldungen.sm_read_ads_parameter := FALSE;
		st_ecd_cmd.meldungen.sm_ec_coe_sdo_write_ex := FALSE;
		st_ecd_cmd.meldungen.sm_ec_coe_sdo_read_ex := FALSE;

		fb_state_entry.i16_next_step := 1;

(*=======================================================*)
	1000: (* Fehler *)
		IF fb_state_entry.E THEN
			st_ecd_cmd.b_job_fehler := TRUE;
			fb_ton_cmd_timeout.IN := FALSE;
			fb_ton_vz.IN := FALSE;
			st_ecd_cmd.enu_cmd := NO_COMMAND;
		END_IF

		(* Fehler reseten *)
		IF st_ecd_cmd.enu_cmd >= ABORT THEN
			st_ecd_cmd.b_job_fehler := FALSE;
			b_jog_vorwaerts_execute := FALSE;
			b_jog_rueckwaerts_execute := FALSE;
			mc_reset_axis.Execute := FALSE;
			mc_home_axis.Execute := FALSE;
			mc_moveabsolute_axis.Execute := FALSE;
			mc_moverelative_axis.Execute := FALSE;
			mc_movevelocity_axis.Execute := FALSE;
			mc_movemodulo_axis.Execute := FALSE;
			mc_setposition_axis.Execute := FALSE;
			mc_halt_axis.Execute := FALSE;
			mc_stop_axis.Execute := FALSE;
			fb_soe_reset.Execute := FALSE;
			fb_soe_write.Execute := FALSE;
			fb_soe_read.Execute := FALSE;
			mc_write_nc_parameter.Execute := FALSE;
			mc_read_nc_parameter.Enable := FALSE;
			fb_ads_write.WRITE := FALSE;
			fb_ads_read.READ := FALSE;
			fb_ec_coe_sdo_write_ex.bExecute := FALSE;
			fb_ec_coe_sdo_read_ex.bExecute := FALSE;
			fb_state_entry.i16_next_step := 0;
		END_IF
END_CASE

(* Endlagenüberwachung der maximalen Verfahrwege der Achse *)
IF b_limitsensor_positiv_vorhanden AND fb_f_trig_limit_sensor_positiv.Q THEN
	mc_stop_axis.Execute := TRUE;
	st_ecd_cmd.meldungen.sm_limit_positiv_erreicht := TRUE;
	fb_state_entry.i16_next_step := 1000;
END_IF
IF b_limitsensor_negativ_vorhanden AND fb_f_trig_limit_sensor_negativ.Q THEN
	mc_stop_axis.Execute := TRUE;
	st_ecd_cmd.meldungen.sm_limit_negativ_erreicht := TRUE;
	fb_state_entry.i16_next_step := 1000;
END_IF

(* Timeout-Fehler aller Drivekommandos *)
IF fb_ton_cmd_timeout.Q THEN
	fb_ton_cmd_timeout.IN := FALSE;
	st_ecd_cmd.meldungen.sm_motion_command_timeout := TRUE;
	fb_state_entry.i16_next_step := 1000;
END_IF

(*Abbruch des aktuellen Achskommandos *)
IF st_ecd_cmd.enu_cmd = ABORT AND fb_state_entry.i16_next_step <> FEHLER THEN
	fb_state_entry.i16_next_step := 999;
END_IF

(* Statehistory *)
fb_state_entry(
	i16_next_step:= ,
	i16_pos:= 2,
	s_debugtext:= ,
	E=> , 
	X=> , 
	i16_step=> ,
	i16_last_step=> );

fb_cmd_history(i16_current_cmd:= st_ecd_cmd.enu_cmd, last_cmd=> );

(*=============================================================================================*)
(* Ab hier werden alle Verfahraufträge für eine Achse abgewickelt *)

(* Lese Zustand der Achse *)
st_masterachse.ReadStatus;

(* Für Rundachsen muss die Sollgeschwindigkeit umgerechnet werden in °/s *)
IF i16_achstyp = RUND OR i16_achstyp = RUND_VIRTUELL THEN
	lr_sollgeschwindigkeit := lr_sollgeschwindigkeit * 360 / 60;
END_IF

(*=============================================================================================*)
(* Reglerfreigabe *)
mc_power_axis(
	Enable:= ,
	Enable_Positive:= ,
	Enable_Negative:= ,
	Override:= lr_override,
	BufferMode:= mc_buffermode_axis,
	Axis:= st_masterachse,
	Status=> ,
	Busy=> ,
	Active=> ,
	Error=> ,
	ErrorID=> );

(*=============================================================================================*)
(* Achse aus Fehlerzustand rücksetzen *)
(* NC-Achse *)
mc_reset_axis(
	Execute:= ,
	Axis:= st_masterachse,
	Done=> ,
	Busy=> ,
	Error=> ,
	ErrorID=> );

(* AX5000 Servokontroller *)
fb_soe_reset(
	NetId:= , 
	Execute:= , 
	Timeout:= t_ads_timeout,
	Axis:= st_masterachse,
	Busy=> ,
	Error=> , 
	AdsErrId=> , 
	SercosErrId=> );

(*=============================================================================================*)
(* Achsposition setzen *)
mc_setposition_axis(
	Execute:= ,
	Position:= st_position.r_soll,
	Mode:= FALSE, (* RELATIVE=True, ABSOLUTE=False (Default) *)
	Options:= ,
	Axis:= st_masterachse,
	Done=> ,
	Busy=> ,
	Error=> ,
	ErrorID=> );

(*=============================================================================================*)
(* Achse referenzieren *)
mc_home_axis(
	Execute:= ,
	Position:= st_position.r_referenz,
	HomingMode:= mc_referenzmodus,
	BufferMode:= mc_buffermode_axis,
	Options:= ,
	bCalibrationCam:= e_referenznocken,
	Axis:= st_masterachse,
	Done=> ,
	Busy=> ,
	Active=> ,
	CommandAborted=> ,
	Error=> ,
	ErrorId=> );

(*=============================================================================================*)
(* Achse tippen *)
mc_jog_axis(
	JogForward:= b_jog_vorwaerts_execute AND NOT b_jog_rueckwaerts_execute,
	JogBackwards:= b_jog_rueckwaerts_execute AND NOT b_jog_vorwaerts_execute,
	Mode:= MC_JOGMODE_CONTINOUS,  (* motion with standard jog parameters for slow motion *)
	Velocity:= lr_sollgeschwindigkeit,
	Acceleration:= st_vorgabe_geschwindigkeiten.lr_beschleunigung,
	Deceleration:= st_vorgabe_geschwindigkeiten.lr_verzoegerung,
	Jerk:= st_vorgabe_geschwindigkeiten.lr_ruck,
	Axis:= st_masterachse,
	Done=> ,
	Busy=> ,
	Active=> ,
	CommandAborted=> ,
	Error=> ,
	ErrorId=> );

(*=============================================================================================*)
(* Fahre Achse absolut *)
mc_moveabsolute_axis(
	Execute:= ,
	Position:= st_position.r_soll,
	Velocity:= lr_sollgeschwindigkeit,
	Acceleration:= st_vorgabe_geschwindigkeiten.lr_beschleunigung,
	Deceleration:= st_vorgabe_geschwindigkeiten.lr_verzoegerung,
	Jerk:= st_vorgabe_geschwindigkeiten.lr_ruck,
	BufferMode:= mc_buffermode_axis,
	Options:= ,
	Axis:= st_masterachse,
	Done=> ,
	Busy=> ,
	Active=> ,
	CommandAborted=> ,
	Error=> ,
	ErrorID=> );
(* Fahre Achse absolut im Falle einer Folgebewegung *)
mc_moveabsolutenext_axis(
	Execute:= ,
	Position:= st_position.r_soll,
	Velocity:= lr_sollgeschwindigkeit,
	Acceleration:= st_vorgabe_geschwindigkeiten.lr_beschleunigung,
	Deceleration:= st_vorgabe_geschwindigkeiten.lr_verzoegerung,
	Jerk:= st_vorgabe_geschwindigkeiten.lr_ruck,
	BufferMode:= mc_buffermode_axis,
	Options:= ,
	Axis:= st_masterachse,
	Done=> ,
	Busy=> ,
	Active=> ,
	CommandAborted=> ,
	Error=> ,
	ErrorID=> );

(*=============================================================================================*)
(* Fahre Achse relaiv *)
mc_moverelative_axis(
	Execute:= ,
	Distance:= st_position.r_soll,
	Velocity:= lr_sollgeschwindigkeit,
	Acceleration:= st_vorgabe_geschwindigkeiten.lr_beschleunigung,
	Deceleration:= st_vorgabe_geschwindigkeiten.lr_verzoegerung,
	Jerk:= st_vorgabe_geschwindigkeiten.lr_ruck,
	BufferMode:= mc_buffermode_axis,
	Options:= ,
	Axis:= st_masterachse,
	Done=> ,
	Busy=> ,
	Active=> ,
	CommandAborted=> ,
	Error=> ,
	ErrorID=> );

(*=============================================================================================*)
(* Gleichlaufachse starten *)
mc_movevelocity_axis(
	Execute:= ,
	Velocity:= lr_sollgeschwindigkeit,
	Acceleration:= st_vorgabe_geschwindigkeiten.lr_beschleunigung,
	Deceleration:= st_vorgabe_geschwindigkeiten.lr_verzoegerung,
	Jerk:= st_vorgabe_geschwindigkeiten.lr_ruck,
	Direction:= mc_richtung_velocity,
	BufferMode:= mc_buffermode_axis,
	Options:= ,
	Axis:= st_masterachse,
	InVelocity=> ,
	Busy=> ,
	Active=> ,
	CommandAborted=> ,
	Error=> ,
	ErrorID=> );

(*=============================================================================================*)
(* Bewegen einer Rundachse *)
mc_movemodulo_axis(
	Execute:= ,
	Position:= st_position.r_soll,
	Velocity:= lr_sollgeschwindigkeit,
	Acceleration:= st_vorgabe_geschwindigkeiten.lr_beschleunigung,
	Deceleration:= st_vorgabe_geschwindigkeiten.lr_verzoegerung,
	Jerk:= st_vorgabe_geschwindigkeiten.lr_ruck,
	Direction:= mc_richtung_modulo,
	BufferMode:= mc_buffermode_axis,
	Options:= ,
	Axis:= st_masterachse,
	Done=> ,
	Busy=> ,
	Active=> ,
	CommandAborted=> ,
	Error=> ,
	ErrorID=> );

(*=============================================================================================*)
mc_stop_axis(
	Execute:= ,
	Deceleration:= st_vorgabe_geschwindigkeiten.lr_verzoegerung,
	Jerk:= st_vorgabe_geschwindigkeiten.lr_ruck,
	Options:= ,
	Axis:= st_masterachse,
	Done=> ,
	Busy=> ,
	Active=> ,
	CommandAborted=> ,
	Error=> ,
	ErrorID=> );

(*=============================================================================================*)
(* MC_Halt führt einen normalen Halt während der Bewegung aus.
Im Gegensatz dazu verriegelt MC_Stop die Achse gegen weitere Bewegungskommandos und
sollte nur in besonderen Situationen angewendet werden. *)
mc_halt_axis(
	Execute:= ,
	Deceleration:= st_vorgabe_geschwindigkeiten.lr_verzoegerung,
	Jerk:= st_vorgabe_geschwindigkeiten.lr_ruck,
	BufferMode:= mc_buffermode_axis,
	Options:= ,
	Axis:= st_masterachse,
	Done=> ,
	Busy=> ,
	Active=> ,
	CommandAborted=> ,
	Error=> ,
	ErrorID=> );

(*=============================================================================================*)
(* Einen Parameter auf den Antrieb schreiben *)
fb_soe_write(
	NetId:= , 
	Idn:= w_idn,	(* Idn := S_0_IDN + 33; *)
	Element:= EC_SOE_ELEMENT_VALUE,
	pSrcBuf:= ADR(ui16_soeparam_write_value),
	BufLen:= SIZEOF(ui16_soeparam_write_value),
	Execute:= , 
	Timeout:= t_ads_timeout,
	Password:= ,
	Axis:= st_masterachse,
	Busy=> ,
	Error=> ,
	AdsErrId=> ,
	SercosErrId=> );

(*=============================================================================================*)
(* Einen Parameter auf dem Antrieb lesen  *)
fb_soe_read(
	NetId:= , 
	Idn:= w_idn,	(* Idn := S_0_IDN + 33; *)
	Element:= EC_SOE_ELEMENT_VALUE,
	pDstBuf:= ADR(ui16_soeparam_read_value),
	BufLen:= SIZEOF(ui16_soeparam_read_value),
	Execute:= , 
	Timeout:= t_ads_timeout,
	Axis:= st_masterachse,
	Busy=> ,
	Error=> , 
	AdsErrId=> ,
	SercosErrId=> , 
	Attribute=> );

(*=============================================================================================*)
(* Einen Parameter auf die NC-Achse schreiben *)
mc_write_nc_parameter(
	Execute:= , 
	ParameterNumber:= i16_nc_parameter_nummer,
	Value:= r_wert_nc_write_parameter,
	Axis:= st_masterachse,
	Done=> ,
	Busy=> ,
	Error=> , 
	ErrorID=> );

(*=============================================================================================*)
(* Einen Parameter von der NC-Achse lesen *)
mc_read_nc_parameter(
	Enable:= , 
	ParameterNumber:= i16_nc_parameter_nummer,
	ReadMode:= READMODE_ONCE,
	Axis:= st_masterachse,
	Valid=> ,
	Busy=> ,
	Error=> , 
	ErrorID=> , 
	Value=> r_wert_nc_read_parameter);

(*=============================================================================================*)
(* Einen beliebigen ADS-Parameter auf die NC-Achse schreiben *)
fb_ads_write(
	NETID:= ,
	PORT:= 501,
	IDXGRP:= st_ads_info.st_symbol_info.idxGroup,
	IDXOFFS:= st_ads_info.st_symbol_info.idxOffset,
	LEN:= st_ads_info.st_symbol_info.byteSize,
	SRCADDR:= st_ads_info.dw_quelladresse_ads_write,
	WRITE:= ,
	TMOUT:= t_ads_timeout,
	BUSY=> , 
	ERR=> , 
	ERRID=> );

(*=============================================================================================*)
(* Einen beliebigen ADS-Parameter von der NC-Achse lesen *)
fb_ads_read(
	NETID:= ,
	PORT:= 501,
	IDXGRP:= st_ads_info.st_symbol_info.idxGroup,
	IDXOFFS:= st_ads_info.st_symbol_info.idxOffset,
	LEN:= st_ads_info.st_symbol_info.byteSize,
	DESTADDR:= st_ads_info.dw_zieladresse_ads_read,
	READ:= , 
	TMOUT:= t_ads_timeout,
	BUSY=> , 
	ERR=> , 
	ERRID=> );

(*=============================================================================================*)
(* Einen neuen EcCoeSdo-Parameter auf den Antrieb schreiben *)
fb_ec_coe_sdo_write_ex(
	sNetId:= st_eccoe_sdo.s_ec_slave_net_id,
	nSlaveAddr:= st_eccoe_sdo.ui16_slave_addr,
	nSubIndex:= st_eccoe_sdo.i8_sub_index,
	nIndex:= st_eccoe_sdo.w_index,
	pSrcBuf:= st_eccoe_sdo.dw_p_source_buffer,
	cbBufLen:= st_eccoe_sdo.ui32_buffer_length,
	bExecute:= ,
	tTimeout:= t_ads_timeout,
	bCompleteAccess:= FALSE,
	bBusy=> , 
	bError=> ,
	nErrId=> );

(*=============================================================================================*)
(* Einen neuen EcCoeSdo-Parameter von dem Antrieb lesen *)
fb_ec_coe_sdo_read_ex(
	sNetId:= st_eccoe_sdo.s_ec_slave_net_id,
	nSlaveAddr:= st_eccoe_sdo.ui16_slave_addr,
	nSubIndex:= st_eccoe_sdo.i8_sub_index,
	nIndex:= st_eccoe_sdo.w_index,
	pDstBuf:= st_eccoe_sdo.dw_p_destination_buffer,
	cbBufLen:= st_eccoe_sdo.ui32_buffer_length,
	bExecute:= ,
	tTimeout:= t_ads_timeout,
	bCompleteAccess:= FALSE,
	bBusy=> ,
	bError=> ,
	nErrId=> );
END_FUNCTION_BLOCK
ACTION sub_TouchProbe:
(*======================================================
   Command: MOVE_TOUCH_PROBE
 ------------------------------------------------------
   Auth: 		Werner Friedl    						 
   Date: 		10.09.2019    						     
   Rev.: 		1.0	
   Desc:		Mit diesem Command kann die Achsposition zu eimem Tastzeitpunkt aufgezeichnet werden.

			- im Achsaufruf müssen diese Einstellungen gemacht werden
		z.B.		b_TriggerInput:=i16_DigitalInput.0		=> Verknüpfung mit den Prozessdaten der Achse an dem der Taster angeklemmt wurde				
				i16_TouchProbeInNo:=1					=> 1 wenn der Taster am Input 1 angeklemmt wurde
				b_SignalEdge:=FallingEdge				=> FallingEdge ODER RisingEdge

		- das Kommando MOVE_TOUCH_PROBE fährt die Achse auf den Taster. Wird der Taster 
			während der Fahrt betätigt , dann stoppt die Achse automatisch und 
			das Messergebniss landet in der VAR lr_RecPos
		
		- Schritt103 => Taster prüfen
		- Schritt104 => Move Absolut und start Touch Probe
		- Schritt105 => Stop Achse und Übergabe Recording Position an die VAR lr_RecPos


		Konfiguration:
		In der IE Hilfe unter "Funktion Probe Unit" findet man die Beschreibung.
		
		im tsm muss der Touch Probe konfiguriert werden.
		Parameter		Wert		
		S-0-0303		405
		S-0-0307		409
		S-0-0169		1
		S-0-0170		3

		in den Prozessdaten einfügen 
		S-0-0801		Digital inputs, sate			und mit der Var i16_DigitalInput der jeweiligen Achse verknüpfen

		im Drivemanager die Logik der Probe unit einstellen 
		- bei Mux1 den Input auswählen und negiert zuweisen
		- 1: Auto activation from SafeOp to Op auswählen

		PLC:
		im VAR_OUTPUT der Achse die Var anlegen
		lr_RecPos							: LREAL;
		
		im VAR anlegen
		i16_DigitalInput						AT %I* : INT;
	
	
		und im Aufruf fb_axis die Var hinzufügen
	
		lr_RecPos=> lr_RecPos,
		b_TriggerInput:=i16_DigitalInput.2,
		b_FallingEdge:=TRUE


 ========================================================*)
IF	mc_touch_probe.Done THEN
	lr_RecPos:=mc_touch_probe.RecordedPosition;
END_IF


(* Touch Probe Initialisierung *)
TriggerInput.EncoderID:= 	st_masterachse.NcToPlc.AxisId;		(* funktioniert so nur wenn die Encoder ID gleich ist wie die Achs ID*)
TriggerInput.TouchProbe:=	TouchProbe1;					(*bei MC_TouchProbe immer TouchProbe1*)
TriggerInput.Edge:=			RisingEdge;						(*bei MC_TouchProbe immer RisingEdge*)
TriggerInput.Mode:=			TOUCHPROBEMODE_SINGLE;



(* Touch Probe Aufruf *)
mc_touch_probe(
	Execute:= ,
	WindowOnly:= 	FALSE ,
	FirstPosition:= ,
	LastPosition:= ,
	Axis:= 			st_masterachse,
	TriggerInput:=	TriggerInput ,
	Done=> ,
	Busy=> ,
	CommandAborted=> ,
	Error=> ,
	ErrorID=> ,
	RecordedPosition=> );

mc_abort_trigger(
	Execute:= ,
	Axis:= 			st_masterachse,
	TriggerInput:=	TriggerInput ,
	Done=> ,
	Busy=> ,
	Error=> , 
	ErrorID=> );
END_ACTION

(* POU EPT Lib/Funktionsbausteine/ST_CommandHistory, ST *)
FUNCTION_BLOCK ST_CommandHistory
VAR_INPUT
	i16_current_cmd 		: enum_ecd_cmd;
END_VAR
VAR_OUTPUT
	last_cmd 			: enum_ecd_cmd;
END_VAR
VAR
	arr_last_cmd_history 	: ARRAY[0..31] OF enum_ecd_cmd;
	i					: INT;
END_VAR
IF (last_cmd <> i16_current_cmd) THEN
	last_cmd := i16_current_cmd;

	FOR i:= 30 TO 0 BY -1DO
		arr_last_cmd_history[i+1] := arr_last_cmd_history[i];
	END_FOR
	arr_last_cmd_history[0] := last_cmd;
END_IF
END_FUNCTION_BLOCK

(* POU EPT Lib/Funktionsbausteine/ST_OT_UT_Ueberwachung, ST *)
FUNCTION_BLOCK ST_OT_UT_Ueberwachung
VAR_INPUT
	lr_achsposition				 : LREAL;
END_VAR
VAR_OUTPUT
	b_error						: BOOL;
END_VAR
VAR
	i32_anfang_ot					: DINT := 0;
	i32_ende_ot					: DINT := 5;
	i32_anfang_ut					: DINT := 180;
	i32_ende_ut					: DINT := 185;
	arr_eintrag					: ARRAY[0..99] OF BOOL := 1,0,1;	(* Länge dient nur zum Nachverfolgen *)
	b_ot							: BOOL := FALSE;
	b_ut							: BOOL := FALSE;
	fb_r_trig_ot					: R_TRIG;
	fb_r_trig_ut					: R_TRIG;
	fb_f_trig_ot					: F_TRIG;
	fb_f_trig_ut					: F_TRIG;
	i							: INT := 0;
END_VAR
(* Kontrollfunktion zum Prüfen, ob auf OT auch immer UT kommt. *)
(* Die Fehlerausgabe erfolgt mittels temporärer Fehlermeldung, welche im Errorlog der Visu mitgeschrieben wird. *)
(* Dies dient der Kontrolle auf fehlbedienung durch das Anlagenpersonal. *)

(* Flanken *)
fb_r_trig_ot(CLK:= b_ot, Q=> );
fb_r_trig_ut(CLK:= b_ut, Q=> );
fb_f_trig_ot(CLK:= b_ot, Q=> );
fb_f_trig_ut(CLK:= b_ut, Q=> );

(* Erstellen der Bereichsnocken *)
IF LREAL_TO_DINT(lr_achsposition) > i32_anfang_ot AND LREAL_TO_DINT(lr_achsposition) < i32_ende_ot THEN
	b_ot := TRUE;
	b_error := FALSE;
ELSE
	b_ot := FALSE;
END_IF

IF LREAL_TO_DINT(lr_achsposition) > i32_anfang_ut AND LREAL_TO_DINT(lr_achsposition) < i32_ende_ut THEN
	b_ut := TRUE;
	b_error := FALSE;
ELSE
	b_ut := FALSE;
END_IF

(* Eintragen von OT bzw. UT in das Register *)
IF fb_r_trig_ot.Q THEN
	FOR i := 99  TO 1 BY -1 DO
		arr_eintrag [i] := arr_eintrag[i - 1];
	END_FOR
	arr_eintrag[0] := 2#0;	(* Eintrag für OT = 0 *)
END_IF

IF fb_r_trig_ut.Q THEN
	FOR i := 99  TO 1 BY -1 DO
		arr_eintrag[i] := arr_eintrag[i - 1];
	END_FOR
	arr_eintrag[0] := 2#1;	(* Eintrag für UT = 1 *)
END_IF

(* Auswertung und Fehler *)
IF fb_f_trig_ot.Q OR fb_f_trig_ut.Q THEN
	b_error := NOT (arr_eintrag[0]  XOR arr_eintrag[1]);
END_IF
END_FUNCTION_BLOCK

(* POU Gemeinsamkeiten17xx/Bedienen/ST_Euchner_Handbedienpult, ST *)
PROGRAM ST_Euchner_Handbedienpult
VAR
	(* Eingänge von der Hardware *)
	e_Taste_Zustimm			AT %I* : BOOL;
	e_Taste_Plus				AT %I* : BOOL;
	e_Taste_Power			AT %I* : BOOL;
	e_Taste_Minus			AT %I* : BOOL;

	e_i16_Zaehler			AT %I* : INT;

	(* Instanzen *)
	fb_ton					: TON;

	(* Merker *)
	i16_merkpos				: INT := 0;
END_VAR
VAR_OUTPUT
	b_Taste_Zustimm			: BOOL := FALSE;
	b_Taste_Plus				: BOOL := FALSE;
	b_Taste_Power			: BOOL := FALSE;
	b_Taste_Minus			: BOOL := FALSE;

	i16_Handrad_delta		: INT := 0;
END_VAR
(* Tasten *)
b_Taste_Zustimm	:= e_Taste_Zustimm;
b_Taste_Plus	:= e_Taste_Plus;
b_Taste_Power := e_Taste_Power;
b_Taste_Minus := e_Taste_Minus;

(* Generiere Impuls für Delta Zähler *)
fb_ton(IN:= NOT fb_ton.Q , PT:= t#100ms, Q=> , ET=> );

IF fb_ton.Q THEN
	i16_Handrad_delta := e_i16_Zaehler - i16_merkpos;
	i16_merkpos := e_i16_Zaehler;
END_IF
END_PROGRAM

(* POU Gemeinsamkeiten17xx/Bedienen/ST_TippTasten, ST *)
PROGRAM ST_TippTasten
VAR_INPUT
	(* Geschwindigkeit / Stufe *)
	i16_akt_stufe						: INT := 0;	(* 0-9 *)
	b_initialisierungsphase				: BOOL := FALSE;
	b_einfaedeln_aktiv				: BOOL := FALSE;
END_VAR
VAR_IN_OUT
	st_visu							: struct_visu;
	st_visu_hinten						: struct_visu_hinten;
END_VAR
VAR
	lr_override						: LREAL := 25;
	lr_override_gestuft					: LREAL := 10;
	r_trig_tippen						: R_TRIG;
	r_trig_tippen_einfaedeln			: R_TRIG;
	r_trig_vorgabe					: R_TRIG;
	b_freigabe_override_auto			: BOOL := FALSE;
	fb_r_trig_quittieren					: R_TRIG;
END_VAR

VAR CONSTANT
	lr_override_init_einfaedel			: LREAL := 25;
END_VAR
(* Mit den zeitlichen Impulsen vom Handrad lässt sich der Override aller Achsen verändern. Die Geschwindigkeit wird im "ST_AxisJobCtrl_Motion" limitiert. *)
(* Tipp-Taste *)

r_trig_tippen(
		CLK:=NOT b_einfaedeln_aktiv AND (st_visu.b_tippen_start OR visu_hinten.out.b_start OR ST_Euchner_Handbedienpult.b_Taste_Power),
		Q=> );
r_trig_tippen_einfaedeln(
		CLK:= b_einfaedeln_aktiv AND (st_visu_hinten.out.b_tippen OR ST_Euchner_Handbedienpult.b_Taste_Power),
		Q=> );
r_trig_vorgabe(
		CLK:= st_visu.b_geschwindigkeit_vorgabe, Q=> );

(* Flanken *)
fb_r_trig_quittieren(CLK:= st_visu.b_quittieren OR st_visu_hinten.out.b_quittieren, Q=> );

CASE gi16_betriebsart OF
	AUTO:
		gb_ba_auto_kontroller := TRUE;

		IF r_trig_tippen.Q OR fb_r_trig_quittieren.Q THEN
			b_freigabe_override_auto := TRUE;
		END_IF

		IF b_einfaedeln_aktiv OR b_initialisierungsphase THEN
			lr_override := lr_override_gestuft := lr_override_init_einfaedel;
		ELSE

			IF r_trig_vorgabe.Q THEN
				i16_akt_stufe := 9;
			END_IF
			IF b_freigabe_override_auto THEN
				(* Override für Achsen mit "Vollgas" im Automatikbetrieb *)
				lr_override := 100;
				(* Override für Achsen, welche in Abstufung gefahren werden *)
				IF  i16_akt_stufe>= 0 AND i16_akt_stufe<= 9 THEN
					(* Overridevorgabe im Automatikbetrieb *)
					lr_override_gestuft := (i16_akt_stufe +1) * 10;
				ELSE
					(* Falls Geschwindigkeitsstufe was anderes als 0-9 enthält: Override auf 0: Keine Achse fährt *)
					lr_override_gestuft := 0;
				END_IF
			ELSE
				lr_override := lr_override_gestuft := 0;
			END_IF
		END_IF

	TIPPEN:
		b_freigabe_override_auto := FALSE;

		IF r_trig_tippen.Q OR lr_override > 0 OR  lr_override_gestuft > 0 THEN
			gb_ba_auto_kontroller := TRUE;
		ELSE
			gb_ba_auto_kontroller := FALSE;
		END_IF

		IF ST_Euchner_Handbedienpult.i16_Handrad_delta > 0 THEN
			lr_override := lr_override_gestuft := ABS(ST_Euchner_Handbedienpult.i16_Handrad_delta) * 0.1;
		ELSE
			lr_override := lr_override_gestuft := 0;
		END_IF

	HAND:
		gb_ba_auto_kontroller := FALSE;
		b_freigabe_override_auto := FALSE;
		lr_override := lr_override_gestuft := ABS(ST_Euchner_Handbedienpult.i16_Handrad_delta)* 0.1;
END_CASE

(* Abfrage maximaler Override grösser 100% *)
IF lr_override > 100 THEN
	lr_override := 100;
END_IF
IF lr_override_gestuft > 100 THEN
	lr_override_gestuft := 100;
END_IF
END_PROGRAM

(* POU Gemeinsamkeiten17xx/Achsen/ST_MotionFunctionPoints, ST *)
PROGRAM ST_MotionFunctionPoints
VAR_INPUT
	st_ctrl_in								: struct_ctrl_in;
END_VAR
VAR_OUTPUT
	st_ctrl_out							: struct_ctrl_out;
END_VAR
VAR
	fb_ton_wz							: TON;
	fb_ton_quitt							: TON;
	fb_state_entry						: ST_StateEntry;
	i, j									: INT := 0;
	udi_table_id_bestueckachse			: UDINT := 0;
	arr_motion_function_points		: ARRAY[1..ARRAY_LAENGE_MFP] OF struct_db_motionfunctionpoint;
END_VAR
VAR CONSTANT
	ARRAY_LAENGE_MFP				: INT := 100;
	YZTischMasterPos2					 : LREAL := 125;
	YZTischMasterPos3					 : LREAL := 185;
END_VAR
(* Zeiten *)
fb_ton_wz(IN:= ,PT:= , Q=>  , ET=> );
fb_ton_quitt(IN:= , PT:= t#50ms, Q=> , ET=> );

(* =====Berechnung MFPs===== *)
(* Berechnung von Punkten in einer Kurvenscheibe und der maximalen Mastergeschwindigkeit *)

(* =====Kopplung: Virtuelle Masterachse <-> Z-Achse ===== *)
fb_edit_mfps_bestuecken_z.fb(
	st_config:= fb_edit_mfps_bestuecken_z.st_config,
	st_ctrl_in:= fb_edit_mfps_bestuecken_z.st_ctrl.in,
	udiTableId:= 1,
	eMotionFunctionType:= MOTIONFUNCTYPE_POLYNOM5,
	i16_startpunkt_edit_mf_tab:= 2,
	arr_db_mf_tab:= arr_motion_function_points,
	lrVeloMax:= ST_Z_Achse.st_geschwindigkeiten.lr_maximalgeschwindigkeit,
	lrAccMax:= ST_Z_Achse.st_geschwindigkeiten.lr_beschleunigung,
	lrDecMax:= ST_Z_Achse.st_geschwindigkeiten.lr_verzoegerung,
	lrModuloValue:= 360.0,
	st_AxisRefMaster:= virtuelle_master_achse,
	st_AxisRefSlave:= z_achse,
	lrMasterVeloMax=> ,		(* Maximum Master Velocity [°/s] *)
	lrMasterRotPerMinMax=> ,	(* Maximum Master Rotations per Minute [1/min] *)
	st_ctrl_out=> fb_edit_mfps_bestuecken_z.st_ctrl.out);

(* =====Kopplung: Virtuelle Masterachse <-> Y-Achse ===== *)
fb_edit_mfps_bestuecken_y.fb(
	st_config:= fb_edit_mfps_bestuecken_y.st_config,
	st_ctrl_in:= fb_edit_mfps_bestuecken_y.st_ctrl.in,
	udiTableId:= 3,
	eMotionFunctionType:= MOTIONFUNCTYPE_POLYNOM5,
	i16_startpunkt_edit_mf_tab:= 2,
	arr_db_mf_tab:= arr_motion_function_points,
	lrVeloMax:= ST_Y_Achse.st_geschwindigkeiten.lr_maximalgeschwindigkeit,
	lrAccMax:= ST_Y_Achse.st_geschwindigkeiten.lr_beschleunigung,
	lrDecMax:= ST_Y_Achse.st_geschwindigkeiten.lr_verzoegerung,
	lrModuloValue:= 360.0,
	st_AxisRefMaster:= virtuelle_master_achse,
	st_AxisRefSlave:= y_achse,
	lrMasterVeloMax=> ,		(* Maximum Master Velocity [°/s] *)
	lrMasterRotPerMinMax=> ,	(* Maximum Master Rotations per Minute [1/min] *)
	st_ctrl_out=> fb_edit_mfps_bestuecken_y.st_ctrl.out);

(* =====Kopplung: Virtuelle Masterachse <-> Servobandeinzug-Achse ===== *)
fb_edit_mfps_bestuecken_b.fb(
	st_config:= fb_edit_mfps_bestuecken_b.st_config,
	st_ctrl_in:= fb_edit_mfps_bestuecken_b.st_ctrl.in,
	udiTableId:= 4,
	eMotionFunctionType:= MOTIONFUNCTYPE_POLYNOM5,
	i16_startpunkt_edit_mf_tab:= 2,
	arr_db_mf_tab:= arr_motion_function_points,
	lrVeloMax:= ST_Servobandeinzug.st_geschwindigkeiten.lr_maximalgeschwindigkeit,
	lrAccMax:= ST_Servobandeinzug.st_geschwindigkeiten.lr_beschleunigung,
	lrDecMax:= ST_Servobandeinzug.st_geschwindigkeiten.lr_verzoegerung,
	lrModuloValue:= 360.0,
	st_AxisRefMaster:= bestueckachse,
	st_AxisRefSlave:= b_achse,
	lrMasterVeloMax=> ,		(* Maximum Master Velocity [°/s] *)
	lrMasterRotPerMinMax=> ,	(* Maximum Master Rotations per Minute [1/min] *)
	st_ctrl_out=> fb_edit_mfps_bestuecken_b.st_ctrl.out);

(* =====Kopplung: Z-Achse <-> Y-Achse ===== *)
fb_edit_mfps_yz_tisch.fb(
	st_config:= fb_edit_mfps_yz_tisch.st_config,
	st_ctrl_in:= fb_edit_mfps_yz_tisch.st_ctrl.in,
	udiTableId:= 2,
	eMotionFunctionType:= MOTIONFUNCTYPE_POLYNOM5,
	i16_startpunkt_edit_mf_tab:= 2,
	arr_db_mf_tab:= arr_motion_function_points,
	lrVeloMax:= ST_Y_Achse.st_geschwindigkeiten.lr_maximalgeschwindigkeit,
	lrAccMax:= ST_Y_Achse.st_geschwindigkeiten.lr_beschleunigung,
	lrDecMax:= ST_Y_Achse.st_geschwindigkeiten.lr_verzoegerung,
	lrModuloValue:= 0.0,
	st_AxisRefMaster:= z_achse,
	st_AxisRefSlave:= y_achse,
	lrMasterVeloMax=> ,		(* Maximum Master Velocity [mm/s] *)
	lrMasterRotPerMinMax=> ,	(* Maximum Master Rotations per Minute [1/min] *)
	st_ctrl_out=> fb_edit_mfps_yz_tisch.st_ctrl.out);

(* =====Kopplung: Virtuelle Masterachse <-> Bestueckachse ===== *)
(*
fb_edit_mfps_bestueckachse.fb(
	st_config:= fb_edit_mfps_bestueckachse.st_config,
	st_ctrl_in:= fb_edit_mfps_bestueckachse.st_ctrl.in,
	udiTableId:= udi_table_id_bestueckachse,
	eMotionFunctionType:= MOTIONFUNCTYPE_POLYNOM5,
	i16_startpunkt_edit_mf_tab:= 1,
	arr_db_mf_tab:= gst_datensatz.st_wkz.st_virtmaster_bestueckachse.arr_motion_function_points,
	lrVeloMax:= ST_Bestueckachse.st_geschwindigkeiten.lr_maximalgeschwindigkeit,
	lrAccMax:= ST_Bestueckachse.st_geschwindigkeiten.lr_beschleunigung,
	lrDecMax:= ST_Bestueckachse.st_geschwindigkeiten.lr_verzoegerung,
	lrModuloValue:= 360.0,
	st_AxisRefMaster:= virtuelle_master_achse,
	st_AxisRefSlave:= bestueckachse,
	lrMasterVeloMax=> ,		(* Maximum Master Velocity [°/s] *)
	lrMasterRotPerMinMax=> ,	(* Maximum Master Rotations per Minute [1/min] *)
	st_ctrl_out=> fb_edit_mfps_bestueckachse.st_ctrl.out);
*)
fb_camtable_bestueckachse.fb(
	st_config:= fb_camtable_bestueckachse.st_config,
	st_ctrl_in:= fb_camtable_bestueckachse.st_ctrl.in,
	udiTableId:= udi_table_id_bestueckachse,
	arr_db_mf_tab:= arr_motion_function_points,
	lrModuloValue:= 360,
	st_AxisRefMaster:= virtuelle_master_achse,
	st_AxisRefSlave:= bestueckachse,
	st_ctrl_out=> fb_camtable_bestueckachse.st_ctrl.out);

(* =======================================Toplevel========================================== *)
IF fb_state_entry.i16_next_step > INIT AND fb_state_entry.i16_next_step < FEHLER THEN
	(* =====Fehler MFP-Berechnung===== *)
	IF 	fb_edit_mfps_bestuecken_z.st_ctrl.out.b_fehler OR
		fb_edit_mfps_bestuecken_y.st_ctrl.out.b_fehler OR
		fb_edit_mfps_bestuecken_b.st_ctrl.out.b_fehler OR
		fb_edit_mfps_yz_tisch.st_ctrl.out.b_fehler OR
		fb_camtable_bestueckachse.st_ctrl.out.b_fehler
		THEN
			fb_state_entry.i16_next_step := FEHLER;
	END_IF

	IF fb_state_entry.i16_next_step < STOP THEN
		IF st_ctrl_in.b_stop THEN
			fb_state_entry.i16_next_step := STOP;
		END_IF
	END_IF
END_IF

(* ======================================Schrittkette======================================== *)
fb_state_entry(
	i16_next_step:= ,
	i16_pos:= 1,
	s_debugtext:= ,
	E=> ,
	X=> ,
	i16_step=> ,
	i16_last_step=> );

CASE fb_state_entry.i16_step OF
	INIT_OBJ:
		fb_state_entry.i16_next_step := INIT;

(*=======================================================*)
	INIT:
		IF fb_state_entry.E THEN
			fb_ton_wz.IN := FALSE;
			fb_ton_quitt.IN := FALSE;
			st_ctrl_out.b_fehler := FALSE;
			st_ctrl_out.b_fertig := FALSE;
			st_ctrl_out.b_bereit := FALSE;

			fb_edit_mfps_bestuecken_z.st_ctrl.in.b_start := FALSE;
			fb_edit_mfps_bestuecken_y.st_ctrl.in.b_start := FALSE;
			fb_edit_mfps_bestuecken_b.st_ctrl.in.b_start := FALSE;
			fb_edit_mfps_yz_tisch.st_ctrl.in.b_start := FALSE;
			fb_camtable_bestueckachse.st_ctrl.in.b_start := FALSE;
		END_IF

		(*-----------------------Weiterschaltbedingungen----------------------------*)
		IF st_ctrl_in.b_init THEN
			fb_edit_mfps_bestuecken_z.st_ctrl.in.b_quitt := FALSE;
			fb_edit_mfps_bestuecken_y.st_ctrl.in.b_quitt := FALSE;
			fb_edit_mfps_bestuecken_b.st_ctrl.in.b_quitt := FALSE;
			fb_edit_mfps_yz_tisch.st_ctrl.in.b_quitt := FALSE;
			fb_camtable_bestueckachse.st_ctrl.in.b_quitt := FALSE;

			CASE gst_datensatz.st_md.i16_typ_zelle OF
				KEINE_ZELLE:
					;

				BESTUECKZELLE_1700:
					fb_state_entry.i16_next_step := 20;

				BESTUECKZELLE_1720:
					fb_state_entry.i16_next_step := 40;

				RASTERFOLIE:
					fb_state_entry.i16_next_step := 50;
			END_CASE
		END_IF

(*===========================MFP berechnen============================*)
	20:	(* Initialisierung der Kurvenscheibenwerte für Bestückachse-ZAchse aus der DB -> grundlegende Definition der Motionfunktion *)
		(* 1700 *)
		IF fb_state_entry.E THEN
			(* Kurvenscheibe Best-Z-Achse *)
			subr_ST_MFP_Z_Achse();
		END_IF

		(*-----------------------Weiterschaltbedingungen----------------------------*)
		IF fb_edit_mfps_bestuecken_z.fb.st_ctrl_out.b_fertig AND NOT fb_state_entry.E THEN
			fb_edit_mfps_bestuecken_z.st_ctrl.in.b_start := FALSE;
			fb_state_entry.i16_next_step := 21;
		END_IF

(*=======================================================*)
	21:	(* 1700 *)
		IF fb_state_entry.E THEN
			(* Kurvenscheibe Best-Y-Achse *)
			subr_ST_MFP_Y_Achse();
		END_IF

		(*-----------------------Weiterschaltbedingungen----------------------------*)
		IF fb_edit_mfps_bestuecken_y.fb.st_ctrl_out.b_fertig AND NOT fb_state_entry.E THEN
			fb_edit_mfps_bestuecken_y.st_ctrl.in.b_start := FALSE;
			fb_state_entry.i16_next_step := 22;
		END_IF

(*=======================================================*)
	22:	(* 1700 *)
		IF fb_state_entry.E THEN
			(* Kurvenscheibe Y-Z-Tisch *)
			subr_ST_MFP_YZ_Tisch();
		END_IF

		(*-----------------------Weiterschaltbedingungen----------------------------*)
		IF fb_edit_mfps_yz_tisch.st_ctrl.out.b_fertig AND NOT fb_state_entry.E THEN
			fb_edit_mfps_yz_tisch.st_ctrl.in.b_start := FALSE;
			fb_state_entry.i16_next_step := 23;
		END_IF

(*=======================================================*)
	23:	(* 1700 *)
		IF fb_state_entry.E THEN
			(* Kurvenscheibe mit Scalierung 1 Virtuelle Masterachse - Bestückachse *)
			subr_ST_MFP_Bestueckachse_S1();
		END_IF

		(*-----------------------Weiterschaltbedingungen----------------------------*)
		IF fb_camtable_bestueckachse.st_ctrl.out.b_fertig AND NOT fb_state_entry.E THEN
			fb_camtable_bestueckachse.st_ctrl.in.b_start := FALSE;
			fb_state_entry.i16_next_step := 24;
		END_IF

(*=======================================================*)
	24:	(* 1700 *)
		IF fb_state_entry.E THEN
			(* Kurvenscheibe mit Scalierung 0 Virtuelle Masterachse - Bestückachse *)
			subr_ST_MFP_Bestueckachse_S0();
		END_IF

		(*-----------------------Weiterschaltbedingungen----------------------------*)
		IF fb_camtable_bestueckachse.st_ctrl.out.b_fertig AND NOT fb_state_entry.E THEN
			fb_camtable_bestueckachse.st_ctrl.in.b_start := FALSE;
			fb_state_entry.i16_next_step := 25;
		END_IF

(*=======================================================*)
	25:	(* 1700 *)
		IF fb_state_entry.E THEN
			CASE gst_datensatz.st_wkz.i16_typ_bandeinzug OF
				BANDWECHSLER_V2:
					fb_state_entry.i16_next_step := BEREIT;
				SERVO:
					(* Kurvenscheibe Best-Servobandeinzug-Achse *)
					subr_ST_MFP_B_Achse();
			END_CASE;
		END_IF

		(*-----------------------Weiterschaltbedingungen----------------------------*)
		IF fb_edit_mfps_bestuecken_b.fb.st_ctrl_out.b_fertig AND NOT fb_state_entry.E THEN
			fb_edit_mfps_bestuecken_b.st_ctrl.in.b_start := FALSE;
			fb_state_entry.i16_next_step := BEREIT;
		END_IF

(*=======================================================*)
	30:	(* Initialisierung der Kurvenscheibenwerte für Bestückachse-ZAchse aus der DB -> grundlegende Definition der Motionfunktion *)
		(* RASTERPLATTE *)
		IF fb_state_entry.E THEN
			(* Kurvenscheibe Y-Z-Tisch *)
			subr_ST_MFP_YZ_Tisch();
		END_IF

		(*-----------------------Weiterschaltbedingungen----------------------------*)
		IF fb_edit_mfps_yz_tisch.st_ctrl.out.b_fertig AND NOT fb_state_entry.E THEN
			fb_edit_mfps_yz_tisch.st_ctrl.in.b_start := TRUE;
			fb_state_entry.i16_next_step := BEREIT;
		END_IF

(*=======================================================*)
	40:	(* Initialisierung der Kurvenscheibenwerte für Bestückachse-ZAchse aus der DB -> grundlegende Definition der Motionfunktion *)
		(* 1720 *)
		IF fb_state_entry.E THEN
			(* Kurvenscheibe Best-Z-Achse *)
			FOR i := 1 TO ARRAY_LAENGE_MFP BY 1DO
				arr_motion_function_points[i].PointIndex := i;
				arr_motion_function_points[i].FunctionType := MOTIONFUNCTYPE_NOTDEF;
				arr_motion_function_points[i].PointType := MOTIONPOINTTYPE_IGNORE;
				arr_motion_function_points[i].MasterPos := 0.0;
				arr_motion_function_points[i].SlavePos := 0.0;
			END_FOR
			FOR i := 1 TO 4 BY 1DO
				arr_motion_function_points[i].PointIndex := i;
				arr_motion_function_points[i].FunctionType := MOTIONFUNCTYPE_POLYNOM1;
				arr_motion_function_points[i].PointType := MOTIONPOINTTYPE_VELOCITY;
			END_FOR
			arr_motion_function_points[2].FunctionType := MOTIONFUNCTYPE_POLYNOM5_MM;
			arr_motion_function_points[1].MasterPos := 0.0;
			arr_motion_function_points[1].SlavePos := 0.0;
			arr_motion_function_points[2].MasterPos := 250;
			arr_motion_function_points[2].SlavePos := 0.0;
			arr_motion_function_points[3].MasterPos := 340;
			arr_motion_function_points[3].SlavePos := 1;
			arr_motion_function_points[4].MasterPos := 360;
			arr_motion_function_points[4].SlavePos := 1;
			fb_edit_mfps_bestuecken_z.st_ctrl.in.b_start := TRUE;
		END_IF

		(*-----------------------Weiterschaltbedingungen----------------------------*)
		IF fb_edit_mfps_bestuecken_z.fb.st_ctrl_out.b_fertig AND NOT fb_state_entry.E THEN
			fb_edit_mfps_bestuecken_z.st_ctrl.in.b_start := FALSE;
			fb_state_entry.i16_next_step := 41;
		END_IF

(*=======================================================*)
	41:	(* 1720 *)
		IF fb_state_entry.E THEN
			(* Kurvenscheibe mit Scalierung 1 Virtuelle Masterachse - Bestückachse *)
			subr_ST_MFP_Bestueckachse_S1();
		END_IF

		(*-----------------------Weiterschaltbedingungen----------------------------*)
		IF fb_camtable_bestueckachse.st_ctrl.out.b_fertig AND NOT fb_state_entry.E THEN
			fb_camtable_bestueckachse.st_ctrl.in.b_start := FALSE;
			fb_state_entry.i16_next_step := 42;
		END_IF

(*=======================================================*)
	42:	(* 1720 *)
		IF fb_state_entry.E THEN
			(* Kurvenscheibe mit Scalierung 0 Virtuelle Masterachse - Bestückachse *)
			subr_ST_MFP_Bestueckachse_S0();
		END_IF

		(*-----------------------Weiterschaltbedingungen----------------------------*)
		IF fb_camtable_bestueckachse.st_ctrl.out.b_fertig AND NOT fb_state_entry.E THEN
			fb_camtable_bestueckachse.st_ctrl.in.b_start := FALSE;
			fb_state_entry.i16_next_step := BEREIT;
		END_IF

(*=======================================================*)
	50:	(* Rasterfolie *)
		IF fb_state_entry.E THEN
			(* Kurvenscheibe Best-Z-Achse *)
			subr_ST_MFP_Z_Achse();
		END_IF

		(*-----------------------Weiterschaltbedingungen----------------------------*)
		IF fb_edit_mfps_bestuecken_z.fb.st_ctrl_out.b_fertig AND NOT fb_state_entry.E THEN
			fb_edit_mfps_bestuecken_z.st_ctrl.in.b_start := FALSE;
			fb_state_entry.i16_next_step := 51;
		END_IF

(*=======================================================*)
	51:	(* Rasterfolie *)
		IF fb_state_entry.E THEN
			(* Kurvenscheibe Best-Y-Achse *)
			subr_ST_MFP_Y_Achse();
		END_IF

		(*-----------------------Weiterschaltbedingungen----------------------------*)
		IF fb_edit_mfps_bestuecken_y.fb.st_ctrl_out.b_fertig AND NOT fb_state_entry.E THEN
			fb_edit_mfps_bestuecken_y.st_ctrl.in.b_start := FALSE;
			fb_state_entry.i16_next_step := 52;
		END_IF

(*=======================================================*)
	52:	(* Rasterfolie *)
		IF fb_state_entry.E THEN
			(* Kurvenscheibe Y-Z-Tisch *)
			FOR i := 1 TO ARRAY_LAENGE_MFP BY 1DO
				arr_motion_function_points[i].PointIndex := i;
				arr_motion_function_points[i].FunctionType := MOTIONFUNCTYPE_NOTDEF;
				arr_motion_function_points[i].PointType := MOTIONPOINTTYPE_IGNORE;
				arr_motion_function_points[i].MasterPos := 0.0;
				arr_motion_function_points[i].SlavePos := 0.0;
			END_FOR
			FOR i := 1 TO 4 BY 1DO
				arr_motion_function_points[i].PointIndex := i;
				arr_motion_function_points[i].FunctionType := MOTIONFUNCTYPE_POLYNOM1;
				arr_motion_function_points[i].PointType := MOTIONPOINTTYPE_VELOCITY;
			END_FOR
			arr_motion_function_points[2].FunctionType := MOTIONFUNCTYPE_POLYNOM5_MM;
			arr_motion_function_points[1].MasterPos := -115;
			arr_motion_function_points[1].SlavePos := gst_datensatz.st_wkz.st_yz_tisch.r_wkz_einfahrpos_y;
			arr_motion_function_points[2].MasterPos := gst_datensatz.st_wkz.st_yz_tisch.r_wkz_einfahrpos_z;
			arr_motion_function_points[2].SlavePos := gst_datensatz.st_wkz.st_yz_tisch.r_wkz_einfahrpos_y;
			arr_motion_function_points[3].MasterPos := 175;
			arr_motion_function_points[3].SlavePos := gst_datensatz.st_md.st_md_y_achse.lr_wt_uebergabepos;
			arr_motion_function_points[4].MasterPos := 200;
			arr_motion_function_points[4].SlavePos := gst_datensatz.st_md.st_md_y_achse.lr_wt_uebergabepos;
			fb_edit_mfps_yz_tisch.st_ctrl.in.b_start := TRUE;
		END_IF

		(*-----------------------Weiterschaltbedingungen----------------------------*)
		IF fb_edit_mfps_yz_tisch.st_ctrl.out.b_fertig AND NOT fb_state_entry.E THEN
			fb_edit_mfps_yz_tisch.st_ctrl.in.b_start := FALSE;
			fb_state_entry.i16_next_step := 53;
		END_IF

(*=======================================================*)
	53:	(* Rasterfolie *)
		IF fb_state_entry.E THEN
			(* Kurvenscheibe mit Scalierung 1 Virtuelle Masterachse - Bestückachse *)
			subr_ST_MFP_Bestueckachse_S1();
		END_IF

		(*-----------------------Weiterschaltbedingungen----------------------------*)
		IF fb_camtable_bestueckachse.st_ctrl.out.b_fertig AND NOT fb_state_entry.E THEN
			fb_camtable_bestueckachse.st_ctrl.in.b_start := FALSE;
			fb_state_entry.i16_next_step := 54;
		END_IF

(*=======================================================*)
	54:	(* Rasterfolie *)
		IF fb_state_entry.E THEN
			(* Kurvenscheibe mit Scalierung 0 Virtuelle Masterachse - Bestückachse *)
			subr_ST_MFP_Bestueckachse_S0();
		END_IF

		(*-----------------------Weiterschaltbedingungen----------------------------*)
		IF fb_camtable_bestueckachse.st_ctrl.out.b_fertig AND NOT fb_state_entry.E THEN
			fb_camtable_bestueckachse.st_ctrl.in.b_start := FALSE;
			fb_state_entry.i16_next_step := BEREIT;
		END_IF

(*=======================================================*)
	BEREIT:
		IF fb_state_entry.E THEN
			st_ctrl_out.b_bereit := TRUE;
		END_IF

(*=======================================================*)
	FEHLER:
		IF fb_state_entry.E THEN
			st_ctrl_out.b_fehler := TRUE;
			fb_ton_quitt.IN := FALSE;
			fb_edit_mfps_bestuecken_z.st_ctrl.in.b_quitt := FALSE;
			fb_edit_mfps_bestuecken_y.st_ctrl.in.b_quitt := FALSE;
			fb_edit_mfps_bestuecken_b.st_ctrl.in.b_quitt := FALSE;
			fb_edit_mfps_yz_tisch.st_ctrl.in.b_quitt := FALSE;
			fb_camtable_bestueckachse.st_ctrl.in.b_quitt := FALSE;
		END_IF

		(*-----------------------Weiterschaltbedingungen----------------------------*)
		IF st_ctrl_in.b_quitt AND NOT fb_state_entry.E THEN
			st_ctrl_out.b_fehler := FALSE;
			fb_ton_quitt.IN := TRUE;
			fb_edit_mfps_bestuecken_z.st_ctrl.in.b_quitt := TRUE;
			fb_edit_mfps_bestuecken_y.st_ctrl.in.b_quitt := TRUE;
			fb_edit_mfps_bestuecken_b.st_ctrl.in.b_quitt := TRUE;
			fb_edit_mfps_yz_tisch.st_ctrl.in.b_quitt := TRUE;
			fb_camtable_bestueckachse.st_ctrl.in.b_quitt := TRUE;
		END_IF

		IF fb_ton_quitt.Q THEN
			fb_ton_quitt.IN := FALSE;
			fb_state_entry.i16_next_step := INIT;
		END_IF

(*=======================================================*)
	STOP:
		IF fb_state_entry.E THEN
			fb_ton_quitt.IN := FALSE;
			fb_edit_mfps_bestuecken_z.st_ctrl.in.b_quitt := FALSE;
			fb_edit_mfps_bestuecken_y.st_ctrl.in.b_quitt := FALSE;
			fb_edit_mfps_bestuecken_b.st_ctrl.in.b_quitt := FALSE;
			fb_edit_mfps_yz_tisch.st_ctrl.in.b_quitt := FALSE;
			fb_camtable_bestueckachse.st_ctrl.in.b_quitt := FALSE;
		END_IF

		(*-----------------------Weiterschaltbedingungen----------------------------*)
		IF st_ctrl_in.b_quitt AND NOT fb_state_entry.E THEN
			fb_ton_quitt.IN := TRUE;
			fb_edit_mfps_bestuecken_z.st_ctrl.in.b_quitt := TRUE;
			fb_edit_mfps_bestuecken_y.st_ctrl.in.b_quitt := TRUE;
			fb_edit_mfps_bestuecken_b.st_ctrl.in.b_quitt := TRUE;
			fb_edit_mfps_yz_tisch.st_ctrl.in.b_quitt := TRUE;
			fb_camtable_bestueckachse.st_ctrl.in.b_quitt := TRUE;
		END_IF

		IF fb_ton_quitt.Q THEN
			fb_ton_quitt.IN := FALSE;
			fb_state_entry.i16_next_step := INIT;
		END_IF
END_CASE

fb_state_entry(
	i16_next_step:= , 
	i16_pos:= 2,
	s_debugtext:= ,
	E=> , 
	X=> , 
	i16_step=> ,
	i16_last_step=> );
END_PROGRAM
ACTION subr_ST_MFP_B_Achse:
(* Kurvenscheibe Best-Servobandeinzug-Achse *)
FOR i := 1 TO ARRAY_LAENGE_MFP BY 1DO
	arr_motion_function_points[i].PointIndex := i;
	arr_motion_function_points[i].FunctionType := MOTIONFUNCTYPE_NOTDEF;
	arr_motion_function_points[i].PointType := MOTIONPOINTTYPE_IGNORE;
	arr_motion_function_points[i].MasterPos := 0.0;
	arr_motion_function_points[i].SlavePos := 0.0;
END_FOR
FOR i := 1 TO 5 BY 1DO
	arr_motion_function_points[i].PointIndex := i;
	arr_motion_function_points[i].FunctionType := MOTIONFUNCTYPE_POLYNOM1;
	arr_motion_function_points[i].PointType := MOTIONPOINTTYPE_VELOCITY;
END_FOR
arr_motion_function_points[2].FunctionType := MOTIONFUNCTYPE_POLYNOM5_MM;
arr_motion_function_points[1].MasterPos := 0.0;
arr_motion_function_points[1].SlavePos := 0.0;
arr_motion_function_points[2].MasterPos := 50;
arr_motion_function_points[2].SlavePos := 0.0;
arr_motion_function_points[3].MasterPos := 100;
arr_motion_function_points[3].SlavePos := 1;
arr_motion_function_points[4].MasterPos := 200;
arr_motion_function_points[4].SlavePos := 1;
arr_motion_function_points[5].MasterPos := 360;
arr_motion_function_points[5].SlavePos := 1;
fb_edit_mfps_bestuecken_b.st_ctrl.in.b_start := TRUE;
END_ACTION
ACTION subr_ST_MFP_Bestueckachse_S0:
(* Kurvenscheibe mit Scalierung 0 Virtuelle Masterachse - Bestückachse *)
udi_table_id_bestueckachse := 6;
FOR i := 1 TO ARRAY_LAENGE_MFP BY 1DO
	arr_motion_function_points[i].PointIndex := i;
	arr_motion_function_points[i].FunctionType := MOTIONFUNCTYPE_NOTDEF;
	arr_motion_function_points[i].PointType := MOTIONPOINTTYPE_IGNORE;
	arr_motion_function_points[i].MasterPos := 0.0;
	arr_motion_function_points[i].SlavePos := 0.0;
END_FOR
FOR i := 1 TO 2 BY 1DO
	arr_motion_function_points[i].PointIndex := i;
	arr_motion_function_points[i].FunctionType := MOTIONFUNCTYPE_POLYNOM1;
	arr_motion_function_points[i].PointType := MOTIONPOINTTYPE_VELOCITY;
END_FOR
arr_motion_function_points[1].MasterPos := 0;
arr_motion_function_points[1].SlavePos := gst_datensatz.st_md.st_md_bestueckachse.lr_startposition;
arr_motion_function_points[2].MasterPos := 360;
arr_motion_function_points[2].SlavePos := gst_datensatz.st_md.st_md_bestueckachse.lr_startposition;
fb_camtable_bestueckachse.st_ctrl.in.b_start := TRUE;
END_ACTION
ACTION subr_ST_MFP_Bestueckachse_S1:
(* Kurvenscheibe mit Scalierung 1 Virtuelle Masterachse - Bestückachse *)
udi_table_id_bestueckachse := 5;
FOR i := 1 TO ARRAY_LAENGE_MFP BY 1DO
	arr_motion_function_points[i].PointIndex := i;
	arr_motion_function_points[i].FunctionType := MOTIONFUNCTYPE_NOTDEF;
	arr_motion_function_points[i].PointType := MOTIONPOINTTYPE_IGNORE;
	arr_motion_function_points[i].MasterPos := 0.0;
	arr_motion_function_points[i].SlavePos := 0.0;
END_FOR
FOR i := 1 TO 2 BY 1DO
	arr_motion_function_points[i].PointIndex := i;
	arr_motion_function_points[i].FunctionType := MOTIONFUNCTYPE_POLYNOM1;
	arr_motion_function_points[i].PointType := MOTIONPOINTTYPE_VELOCITY;
END_FOR
arr_motion_function_points[1].MasterPos := 0;
arr_motion_function_points[1].SlavePos := 0;
arr_motion_function_points[2].MasterPos := 360;
arr_motion_function_points[2].SlavePos := 360;
fb_camtable_bestueckachse.st_ctrl.in.b_start := TRUE;
END_ACTION
ACTION subr_ST_MFP_Y_Achse:
(* Kurvenscheibe Best-Y-Achse *)
FOR i := 1 TO ARRAY_LAENGE_MFP BY 1DO
	arr_motion_function_points[i].PointIndex := i;
	arr_motion_function_points[i].FunctionType := MOTIONFUNCTYPE_NOTDEF;
	arr_motion_function_points[i].PointType := MOTIONPOINTTYPE_IGNORE;
	arr_motion_function_points[i].MasterPos := 0.0;
	arr_motion_function_points[i].SlavePos := 0.0;
END_FOR
FOR i := 1 TO 4 BY 1DO
	arr_motion_function_points[i].PointIndex := i;
	arr_motion_function_points[i].FunctionType := MOTIONFUNCTYPE_POLYNOM1;
	arr_motion_function_points[i].PointType := MOTIONPOINTTYPE_VELOCITY;
END_FOR
arr_motion_function_points[2].FunctionType := MOTIONFUNCTYPE_POLYNOM5_MM;
arr_motion_function_points[1].MasterPos := 0.0;
arr_motion_function_points[1].SlavePos := 0.0;
arr_motion_function_points[2].MasterPos := 40;
arr_motion_function_points[2].SlavePos := 0.0;
arr_motion_function_points[3].MasterPos := 260;
arr_motion_function_points[3].SlavePos := 1;
arr_motion_function_points[4].MasterPos := 360;
arr_motion_function_points[4].SlavePos := 1;
fb_edit_mfps_bestuecken_y.st_ctrl.in.b_start := TRUE;
END_ACTION
ACTION subr_ST_MFP_YZ_Tisch:
(* Kurvenscheibe Y-Z-Tisch *)


	CASE gst_datensatz.st_md.i16_typ_zelle OF
			KEINE_ZELLE:
					;

			BESTUECKZELLE_1700, BESTUECKZELLE_1720, RASTERFOLIE:

				FOR i := 1 TO ARRAY_LAENGE_MFP BY 1DO
					arr_motion_function_points[i].PointIndex := i;
					arr_motion_function_points[i].FunctionType := MOTIONFUNCTYPE_NOTDEF;
					arr_motion_function_points[i].PointType := MOTIONPOINTTYPE_IGNORE;
					arr_motion_function_points[i].MasterPos := 0.0;
					arr_motion_function_points[i].SlavePos := 0.0;
				END_FOR
				FOR i := 1 TO 4 BY 1DO
					arr_motion_function_points[i].PointIndex := i;
					arr_motion_function_points[i].FunctionType := MOTIONFUNCTYPE_POLYNOM1;
					arr_motion_function_points[i].PointType := MOTIONPOINTTYPE_VELOCITY;
				END_FOR

				IF gst_datensatz.st_wkz.b_variable_einfahrposition THEN
					arr_motion_function_points[2].FunctionType := MOTIONFUNCTYPE_POLYNOM5_MM;
					arr_motion_function_points[1].MasterPos := -115;
					arr_motion_function_points[1].SlavePos := gst_datensatz.st_wkz.st_yz_tisch.r_wkz_einfahrpos_y;
					arr_motion_function_points[2].MasterPos :=gst_datensatz.st_wkz.st_yz_tisch.r_wkz_einfahrpos_z;
					arr_motion_function_points[2].SlavePos := gst_datensatz.st_wkz.st_yz_tisch.r_wkz_einfahrpos_y;
					arr_motion_function_points[3].MasterPos := YZTischMasterPos3;
					arr_motion_function_points[3].SlavePos := gst_datensatz.st_md.st_md_y_achse.lr_wt_uebergabepos;
					arr_motion_function_points[4].MasterPos := 200;
					arr_motion_function_points[4].SlavePos := gst_datensatz.st_md.st_md_y_achse.lr_wt_uebergabepos;
				ELSE
					arr_motion_function_points[2].FunctionType := MOTIONFUNCTYPE_POLYNOM5_MM;
					arr_motion_function_points[1].MasterPos := -115;
					arr_motion_function_points[1].SlavePos := gst_datensatz.st_wkz.st_yz_tisch.r_wkz_einfahrpos_y;
					arr_motion_function_points[2].MasterPos := YZTischMasterPos2;
					arr_motion_function_points[2].SlavePos := gst_datensatz.st_wkz.st_yz_tisch.r_wkz_einfahrpos_y;
					arr_motion_function_points[3].MasterPos := YZTischMasterPos3;
					arr_motion_function_points[3].SlavePos := gst_datensatz.st_md.st_md_y_achse.lr_wt_uebergabepos;
					arr_motion_function_points[4].MasterPos := 200;
					arr_motion_function_points[4].SlavePos := gst_datensatz.st_md.st_md_y_achse.lr_wt_uebergabepos;
				END_IF
				fb_edit_mfps_yz_tisch.st_ctrl.in.b_start := TRUE;


	END_CASE
END_ACTION
ACTION subr_ST_MFP_Z_Achse:
(* Kurvenscheibe Best-Z-Achse *)
FOR i := 1 TO ARRAY_LAENGE_MFP BY 1DO
	arr_motion_function_points[i].PointIndex := i;
	arr_motion_function_points[i].FunctionType := MOTIONFUNCTYPE_NOTDEF;
	arr_motion_function_points[i].PointType := MOTIONPOINTTYPE_IGNORE;
	arr_motion_function_points[i].MasterPos := 0.0;
	arr_motion_function_points[i].SlavePos := 0.0;
END_FOR
FOR i := 1 TO 4 BY 1DO
	arr_motion_function_points[i].PointIndex := i;
	arr_motion_function_points[i].FunctionType := MOTIONFUNCTYPE_POLYNOM1;
	arr_motion_function_points[i].PointType := MOTIONPOINTTYPE_VELOCITY;
END_FOR
arr_motion_function_points[2].FunctionType := MOTIONFUNCTYPE_POLYNOM5_MM;
arr_motion_function_points[1].MasterPos := 0.0;
arr_motion_function_points[1].SlavePos := 0.0;
arr_motion_function_points[2].MasterPos := 40;
arr_motion_function_points[2].SlavePos := 0.0;
arr_motion_function_points[3].MasterPos := 260;
arr_motion_function_points[3].SlavePos := 1;
arr_motion_function_points[4].MasterPos := 360;
arr_motion_function_points[4].SlavePos := 1;
fb_edit_mfps_bestuecken_z.st_ctrl.in.b_start := TRUE;
END_ACTION

(* POU Gemeinsamkeiten17xx/Achsen/ST_Z_Achse, ST *)
PROGRAM ST_Z_Achse
VAR_INPUT
	st_config_achse						: struct_ecd_config;
	st_ctrl_in								: struct_ctrl_in;
	e_steuerung_ein						: BOOL;
	e_ba_mit_bedingungen				: BOOL;
	e_tuere_vorne_offen					: BOOL;
	e_tuere_hinten_offen					: BOOL;

	b_start_in							: BOOL;
	lr_Achspos_in						: LREAL;
	lr_Velo_in							: LREAL;
	enu_cmd_in							: enum_ecd_cmd;
END_VAR
VAR_IN_OUT
	st_visu								: struct_ecd_visu;
END_VAR
VAR_OUTPUT
	st_ctrl_out							: struct_ctrl_out;
	t_Z_Achse_ausfahren				: TIME := t#0ms;
	t_Bestueckung					: TIME := t#0ms;
	t_Z_Achse_einfahren				: TIME := t#0ms;
	lr_RecPos						: LREAL;
END_VAR
VAR
	st_sm						 		: struct_ecd_meldungen;
	st_drive_cmd							: struct_ecd_cmd;
	st_drive_cmd_y_achse					: struct_ecd_cmd;
	fb_ton_wz							: TON;
	fb_ton_quitt							: TON;
	fb_ton_wz_disable						: TON;
	fb_ton_taktzeitmessung_wt_wechsel		: TON;
	fb_ton_taktzeitmessung_bestuecken		: TON;
	fb_r_trig_tippen						: R_TRIG;
	fb_f_trig_tippen						: F_TRIG;
	fb_r_trig_taste_plus					: R_TRIG;
	fb_r_trig_start							: R_TRIG;
	fb_r_trig_start_in						: R_TRIG;
	fb_r_trig_hand_dialog					: R_TRIG;
	fb_r_trig_nullpunkt_setzen				: R_TRIG;
	fb_axis								: ST_AxisJobCtrl_Motion;
	fb_axis_y_achse						: ST_AxisJobCtrl_Cam_Gear;
	fb_state_entry							: ST_StateEntry;
	fb_ton_uez							: TON;
	i									: DINT := 0;
	k									: DINT := 0;
	lr_pos_ohneverschiebung			: LREAL;
	fb_r_trig_limit_sensor_positiv			: R_TRIG;
	fb_r_trig_limit_sensor_negativ			: R_TRIG;
	fb_r_trig_skalierungsnocken				: R_TRIG;
	lr_slave_position						: LREAL := 0.0;
	i16_auftrag_cameditor					: enum_auftrag_cameditor;
	i16_kollisionszaehler					: INT := 0;
	b_hand_dialog_aktiv					: BOOL := FALSE;
	b_all_state_parts_ok					: BOOL := FALSE;
	b_kommt_von_init						: BOOL := FALSE;
	i32_UsedTool						: DINT := 0;

	sm_positionsueberwachung				: BOOL := FALSE;
	sm_werkzeugreihenfolge_nicht_io		: BOOL := FALSE;
	sm_keine_bandfreigabe				: BOOL := FALSE;
	sm_tagnummer_ungueltig				: BOOL := FALSE;
	sm_typ_bestueckprogramm_falsch	: BOOL := FALSE;
	sm_keine_rafo_im_einzug		: BOOL := FALSE;


	bm_kein_Pin_im_BB				: BOOL := FALSE;

	(* Kurvenscheibeneditor *)
	i16_startpunkt_mf_tab					: INT := 0;

	st_geschwindigkeiten					: struct_ecd_geschwindigkeiten;
	e_referenz_sensor						AT %I* : BOOL;
	i16_torque							AT %I* : INT;
	i16_DigitalInput						AT %I* : INT;

	lr_vmax_festo							: LREAL := 100.0;

	lr_ReduzierungOverride				: LREAL := 1.0;

	zeit_wt_wechsel						: DINT := 0;
	zeit_wt_bestuecken					: DINT := 0;

	fb_Z_Achse_einfahren			: ST_Taktzeit;
	fb_Bestueckung					: ST_Taktzeit;
	fb_Z_Achse_ausfahren	: ST_Taktzeit;

	lr_decceleration_nothalt				: LREAL;
	lr_decceleration_normal				: LREAL;

	i32_anzahl_rasterfolie				: DINT := 0;

	b_rastnase_vorhanden_vorne			: BOOL;
	b_rastnase_vorhanden_hinten			: BOOL;
	bm_rastnasen_1_fehlt					: BOOL;
	bm_rastnasen_2_fehlt					: BOOL;
	e_kontrolle_rastnase 			AT %I* : BOOL;
	b_teach_pruef_pos1					: BOOL;
	b_teach_pruef_pos2					: BOOL;

	i16_state_msg						: INT;
	Teile_nach_Bandwechsel				: BOOL;
	fb_r_trig_Bandwechsel					: R_TRIG;

	lr_MaxSoftPosLimit					:LREAL;
	lr_MinSoftPosLimit						:LREAL;
	b_EndlageErreicht						:BOOL;
	fb_r_trig_Endlage						: R_TRIG;
	i16_state_msg2						: INT;
END_VAR
(* Die Z-Achse ist der Masterablauf. Sie "weis" wann es losgeht und kennt das Bestückbild.
 * Die Z-Achse schaltet die Bestückachse als Master der Kurvenscheibe ein und startet diese. *)

(* Zeiten *)
fb_ton_wz(IN:= , PT:= , Q=>  , ET=> );
fb_ton_uez(IN:= , PT:= , Q=>  , ET=> );
fb_ton_quitt(IN:= , PT:= t#100ms, Q=> , ET=> );
fb_ton_wz_disable(IN:= , PT:= t#500ms, Q=> , ET=> );

fb_ton_taktzeitmessung_wt_wechsel(IN:= , PT:= t#2h, Q=> , ET=> );
fb_ton_taktzeitmessung_bestuecken(IN:= , PT:= t#2h, Q=> , ET=> );

(*Taktzeitmessung*)
fb_Z_Achse_einfahren(b_start:= , t_zeit=> );
fb_Bestueckung(b_start:= , t_zeit=> );
fb_Z_Achse_ausfahren(b_start:= , t_zeit=> );

(* Flanken *)
fb_r_trig_limit_sensor_positiv(CLK:= st_config_achse.b_limitsensor_positiv_vorhanden AND NOT fb_axis.e_limit_sensor_positive, Q=> );
fb_r_trig_limit_sensor_negativ(CLK:= st_config_achse.b_limitsensor_negativ_vorhanden AND NOT fb_axis.e_limit_sensor_negative, Q=> );
fb_r_trig_taste_plus(CLK:= ST_Euchner_Handbedienpult.b_Taste_Plus, Q=> );
fb_r_trig_start(CLK:= st_ctrl_in.b_start, Q=> );
fb_r_trig_start_in(CLK:= b_start_in, Q=> );
fb_r_trig_skalierungsnocken(CLK:= nockenschaltwerk_bestueckachse.fb.arr_spur[SP_START_SKALIERUNG], Q=> );
fb_r_trig_hand_dialog(CLK:= b_hand_dialog_aktiv, Q=> );
fb_r_trig_nullpunkt_setzen(CLK:=axis_z_achse.st_visu.b_nullpunkt_setzen);

(* Berechnung Override Reduzierung wenn Y-Achse die Rampe fahren muss *)
IF 	gst_datensatz.st_wkz.bFahreSofortAufUebergabePosition AND
	((z_achse.NcToPlc.ActPos > gst_datensatz.st_wkz.st_yz_tisch.r_wkz_einfahrpos_z - 20 AND
	gst_datensatz.st_wkz.b_variable_einfahrposition) OR
	(z_achse.NcToPlc.ActPos > ST_MotionFunctionPoints.YZTischMasterPos2 - 20 AND
	NOT gst_datensatz.st_wkz.b_variable_einfahrposition)) THEN
	lr_ReduzierungOverride := gst_datensatz.st_wkz.r_auto_z / st_geschwindigkeiten.lr_auto_max;
ELSE
	lr_ReduzierungOverride := 1;

END_IF


(*Meldung Teile nach Bandwechsel*)
fb_r_trig_Bandwechsel(CLK:= Teile_nach_Bandwechsel , Q=> );
IF fb_r_trig_Bandwechsel.Q  THEN
	i16_state_msg := 1;
END_IF

(*Produktionsmeldung für Übergabe zu lange*)
CASE i16_state_msg OF
	1: (*Warten bis keine ander Produktions Meldung ansteht *)
		IF	TestAndSet(ST_Message_Produktion.LockFlag) THEN
			ST_Message_Produktion.ClearMessageLines();
			i16_state_msg := 2;
		END_IF

	2:  (*Produktions Meldung*)
		Visu.MeldungProduktion.Color_R := 255;
		Visu.MeldungProduktion.Color_G := 255;
		Visu.MeldungProduktion.Color_B := 0;
		IF visu.s_akt_sprache = 'de' THEN
			Visu.MeldungProduktion.Name:=('Teile nach Bandwechsel');
		ELSIF visu.s_akt_sprache = 'en' THEN
			Visu.MeldungProduktion.Name:=('Teile nach Bandwechsel');
		ELSIF visu.s_akt_sprache = 'cz' THEN
			Visu.MeldungProduktion.Name:=('Teile nach Bandwechsel');
		END_IF
		Visu.MeldungProduktion.ShowMessage := TRUE;
		Visu.MeldungProduktion.Button1.sichtbar:=TRUE;	(*OK*)
		Visu.MeldungProduktion.Button1.Text:='Ok';
		i16_state_msg := 3;

	3:  (*Warte auf OK*)
		IF Visu.MeldungProduktion.Button1.tasten THEN
			i16_state_msg:=0;
		END_IF
END_CASE


(* Achse steuern *)
fb_axis(
	e_referenznocken:= ,
	b_refsensor_vorhanden:= st_config_achse.b_refsensor_vorhanden,
	b_limitsensor_positiv_vorhanden:= st_config_achse.b_limitsensor_positiv_vorhanden,
	b_limitsensor_negativ_vorhanden:= st_config_achse.b_limitsensor_negativ_vorhanden,
	i16_achstyp := st_config_achse.i16_achstyp,
	lr_override_vorgabe:= ST_TippTasten.lr_override * lr_ReduzierungOverride,
	st_position:= ,
	mc_richtung_modulo:= ,
	mc_richtung_velocity:= ,
	mc_referenzmodus:= ,
	mc_buffermode_axis:= ,
	ui16_soeparam_write_value:= ,
	w_idn:= ,
	i16_nc_parameter_nummer:= ,
	r_wert_nc_write_parameter:= ,
	st_vorgabe_geschwindigkeiten:= st_geschwindigkeiten,
	lr_soll_geschwindigkeit:= ,
	b_bedingung_sls:= NOT e_tuere_vorne_offen OR NOT e_tuere_hinten_offen,
	st_ads_info := ,
	st_eccoe_sdo := ,
	st_masterachse:= z_achse,
	st_visu_axis:= st_visu,
	st_ecd_cmd:= st_drive_cmd,
	ui16_soeparam_read_value=> ,
	r_wert_nc_read_parameter=> ,
	lr_RecPos=> lr_RecPos,
	b_TriggerInput:=i16_DigitalInput.1, (*1*)
	b_FallingEdge:=TRUE);

CASE gst_datensatz.st_md.i16_typ_zelle OF
	KEINE_ZELLE:
		;

	BESTUECKZELLE_1700:
		IF gi16_betriebsart = HAND THEN
			(* Bei manuellem Fahren der Slaveachse, muss diese erst entkoppelt werden *)
			IF ST_Y_Achse.b_hand_dialog_aktiv AND y_achse.NcToPlc.CoupleState > 0 THEN
				st_drive_cmd_y_achse.enu_cmd := CAM_OUT_SLAVE;
			END_IF
			(* Achse mit dem Euchner Handbediengerät vorwärts und rückwärts Bewegen*)
			IF fb_r_trig_hand_dialog.Q THEN
				IF y_achse.NcToPlc.CoupleState > 0 THEN
					st_drive_cmd_y_achse.enu_cmd := CAM_OUT_SLAVE;
				END_IF
				fb_state_entry.i16_next_step := HANDRAD;
			END_IF
		END_IF

		IF y_achse.NcToPlc.CoupleState > 0 OR st_drive_cmd_y_achse.enu_cmd > NO_COMMAND THEN
			(* Kurvenscheibenkopplung ein/ausschalten *)
			fb_axis_y_achse(
				r_getriebefaktor:= ,
				r_master_position:= ,
				mc_activation_mode_camin:= ,
				lr_activation_position_camin:= ,
				mc_activation_mode_scaleing:= ,
				lr_activation_position_scaleing:= ,
				mc_buffermode_axis:= ,
				mc_cam_table_id:= 2 ,
				mc_cam_point_id:= ,
				mc_motion_function_point:= ,
				st_camin_options:= ,
				st_camexchange_options:= ,
				mc_reference_cam_table_id:= ,
				st_camscaling_data:= ,
				st_masterachse:= z_achse,
				st_slaveachse:= y_achse,
				st_ecd_cmd:= st_drive_cmd_y_achse );
		END_IF

	BESTUECKZELLE_1720:
		IF gi16_betriebsart = HAND THEN
			(* Achse mit dem Euchner Handbediengerät vorwärts und rückwärts Bewegen*)
			IF fb_r_trig_hand_dialog.Q THEN
				fb_state_entry.i16_next_step := HANDRAD;
			END_IF
		END_IF

	RASTERFOLIE:
		IF gi16_betriebsart = HAND THEN
			(* Bei manuellem Fahren der Slaveachse, muss diese erst entkoppelt werden *)
			IF ST_Y_Achse.b_hand_dialog_aktiv AND y_achse.NcToPlc.CoupleState > 0 THEN
				st_drive_cmd_y_achse.enu_cmd := CAM_OUT_SLAVE;
			END_IF
			(* Achse mit dem Euchner Handbediengerät vorwärts und rückwärts Bewegen*)
			IF fb_r_trig_hand_dialog.Q THEN
				IF y_achse.NcToPlc.CoupleState = 3 THEN
					st_drive_cmd_y_achse.enu_cmd := CAM_OUT_SLAVE;
				END_IF
				fb_state_entry.i16_next_step := HANDRAD;
			END_IF
		END_IF

		IF y_achse.NcToPlc.CoupleState > 0 OR st_drive_cmd_y_achse.enu_cmd > NO_COMMAND THEN
			(* Kurvenscheibenkopplung ein/ausschalten *)
			fb_axis_y_achse(
				r_getriebefaktor:= ,
				r_master_position:= ,
				mc_activation_mode_camin:= ,
				lr_activation_position_camin:= ,
				mc_activation_mode_scaleing:= ,
				lr_activation_position_scaleing:= ,
				mc_buffermode_axis:= ,
				mc_cam_table_id:= 2 ,
				mc_cam_point_id:= ,
				mc_motion_function_point:= ,
				st_camin_options:= ,
				st_camexchange_options:= ,
				mc_reference_cam_table_id:= ,
				st_camscaling_data:= ,
				st_masterachse:= z_achse,
				st_slaveachse:= y_achse,
				st_ecd_cmd:= st_drive_cmd_y_achse );
		END_IF
END_CASE


IF gi16_betriebsart = HAND THEN
	(* Button in der Oberfläche zum setzen des Nullpunktes *)
	IF fb_r_trig_nullpunkt_setzen.Q THEN
		fb_state_entry.i16_next_step :=	NULLPUNKT_SETZEN;
	END_IF
END_IF

(*Meldung Achse hat Endlage überfahren*)
IF lr_MaxSoftPosLimit<>0 AND
  lr_MaxSoftPosLimit < gst_datensatz.st_md.st_md_z_achse.lr_wt_uebergabepos  THEN
	b_EndlageErreicht:= TRUE;
ELSE
	b_EndlageErreicht:=FALSE;
END_IF

fb_r_trig_Endlage(CLK:= b_EndlageErreicht , Q=> );

IF fb_r_trig_Endlage.Q THEN
	i16_state_msg2 := 1;
END_IF

(*Produktionsmeldung für Endlage überfahren*)
CASE i16_state_msg2 OF
	1: (*Warten bis keine ander Produktions Meldung ansteht *)
		IF	TestAndSet(ST_Message_Produktion.LockFlag) THEN
			ST_Message_Produktion.ClearMessageLines();
			i16_state_msg2 := 2;
		END_IF

	2:  (*Produktions Meldung*)
		Visu.MeldungProduktion.Color_R := 255;
		Visu.MeldungProduktion.Color_G := 255;
		Visu.MeldungProduktion.Color_B := 0;
		IF visu.s_akt_sprache = 'de' THEN
			Visu.MeldungProduktion.Name:='Z-Achse WT Übergabepos größer als Endlage';
		ELSIF visu.s_akt_sprache = 'en' THEN
			Visu.MeldungProduktion.Name:='Z-Achse WT Übergabepos größer als Endlage';
		ELSIF visu.s_akt_sprache = 'cz' THEN
			Visu.MeldungProduktion.Name:='Z-Achse WT Übergabepos größer als Endlage';
		END_IF
		Visu.MeldungProduktion.ShowMessage := TRUE;
		Visu.MeldungProduktion.Button1.sichtbar:=FALSE;	(*OK*)
		Visu.MeldungProduktion.Button1.Text:='Ok';
		i16_state_msg2 := 3;

	3:  (*Warte auf OK*)
		IF NOT b_EndlageErreicht THEN
			ST_Message_Produktion.b_PM_Quitt:=TRUE;
			i16_state_msg2:=0;
		END_IF
END_CASE


(* =======================================Toplevel========================================== *)
(* Starte Inbetriebnahme-Sequenz *)
IF st_ctrl_in.b_gehe_step_ibn THEN
	fb_state_entry.i16_next_step := INBETRIEBNAHME;
END_IF

(* =====Achse wird disabled===== *)
IF (NOT e_steuerung_ein OR NOT e_ba_mit_bedingungen) AND z_achse.Status.Operational THEN
	st_drive_cmd.enu_cmd := POWER_DISABLE;
END_IF

IF fb_state_entry.i16_next_step > INIT AND fb_state_entry.i16_next_step < FEHLER THEN
	(* =====Fehler vom Achskontroller===== *)
	IF st_drive_cmd.b_job_fehler OR st_drive_cmd_y_achse.b_job_fehler THEN
		fb_state_entry.i16_next_step := FEHLER;
	END_IF

	IF fb_state_entry.i16_next_step > 40 THEN
		(* Devicefehler *)
		IF z_achse.Status.Error THEN
			st_sm.b_achsfehler := TRUE;
			fb_state_entry.i16_next_step := FEHLER;
		ELSIF z_achse.Status.DriveDeviceError THEN
			st_sm.b_devicefehler := TRUE;
			fb_state_entry.i16_next_step := FEHLER;
		END_IF
	END_IF

	IF fb_state_entry.i16_next_step < STOP THEN
		(* =====Achse wird gestoppt===== *)
		IF st_ctrl_in.b_stop THEN
			fb_state_entry.i16_next_step := STOP;
		ELSIF fb_state_entry.i16_next_step < HALT THEN
			(* =====Achse wird angehalten===== *)
			IF st_ctrl_in.b_halt THEN
				fb_state_entry.i16_next_step := HALT;
			END_IF
		END_IF
	END_IF
END_IF

(* ======================================Schrittkette======================================== *)
fb_state_entry(
	i16_next_step:= , 
	i16_pos:= 1,
	s_debugtext:= ,
	E=> ,
	X=> ,
	i16_step=> ,
	i16_last_step=> );

CASE fb_state_entry.i16_step OF
(*=======================================================*)
	INIT_OBJ:
		IF st_config_achse.b_config_fertig THEN
			fb_state_entry.i16_next_step := 1;
		END_IF

(*=======================================================*)
	1:	(* Warte bis NetID´s der Slaves ausgelesen sind *)
		IF fb_state_entry.E THEN
			;
		END_IF

		(*-----------------------Weiterschaltbedingungen----------------------------*)
		IF ST_EthercatDiag.st_ctrl_out.b_fertig THEN
			fb_state_entry.i16_next_step := 2;
		END_IF

(*=======================================================*)
	2:	(* Spezifische NC-Achsparameter auslesen *)
		IF fb_state_entry.E THEN
			fb_axis.i16_nc_parameter_nummer := MaxVelocitySystem;
			st_drive_cmd.enu_cmd := READ_NC_PARAMETER;
		END_IF

		(*-----------------------Weiterschaltbedingungen----------------------------*)
		IF st_drive_cmd.enu_cmd = NO_COMMAND THEN
			lr_Velo_in:=st_geschwindigkeiten.lr_maximalgeschwindigkeit;
			st_geschwindigkeiten.lr_auto_max := st_geschwindigkeiten.lr_maximalgeschwindigkeit := fb_axis.r_wert_nc_read_parameter;
			st_geschwindigkeiten.lr_auto_min := 50;
			st_geschwindigkeiten.lr_jog := 100;
			fb_state_entry.i16_next_step := 3;
		END_IF

(*=======================================================*)
	3:	(* Spezifische NC-Achsparameter auslesen *)
		IF fb_state_entry.E THEN
			fb_axis.i16_nc_parameter_nummer := MaxAccelerationSystem;
			st_drive_cmd.enu_cmd := READ_NC_PARAMETER;
		END_IF

		(*-----------------------Weiterschaltbedingungen----------------------------*)
		IF st_drive_cmd.enu_cmd = NO_COMMAND THEN
			st_geschwindigkeiten.lr_beschleunigung := fb_axis.r_wert_nc_read_parameter;
			fb_state_entry.i16_next_step := 4;
		END_IF

(*=======================================================*)
	4:	(* Spezifische NC-Achsparameter auslesen *)
		IF fb_state_entry.E THEN
			fb_axis.i16_nc_parameter_nummer := MaxDecelerationSystem;
			st_drive_cmd.enu_cmd := READ_NC_PARAMETER;
		END_IF

		(*-----------------------Weiterschaltbedingungen----------------------------*)
		IF st_drive_cmd.enu_cmd = NO_COMMAND THEN
			st_geschwindigkeiten.lr_verzoegerung := fb_axis.r_wert_nc_read_parameter;
			lr_decceleration_normal := st_geschwindigkeiten.lr_verzoegerung;
			lr_decceleration_nothalt := 200000.0;
			fb_state_entry.i16_next_step := 5;
		END_IF

(*=======================================================*)
	5:	(* Spezifische NC-Achsparameter auslesen *)
		IF fb_state_entry.E THEN
			fb_axis.i16_nc_parameter_nummer := MaxJerk;
			st_drive_cmd.enu_cmd := READ_NC_PARAMETER;
		END_IF

		(*-----------------------Weiterschaltbedingungen----------------------------*)
		IF st_drive_cmd.enu_cmd = NO_COMMAND THEN
			st_geschwindigkeiten.lr_ruck := fb_axis.r_wert_nc_read_parameter;
			fb_state_entry.i16_next_step := 6;
		END_IF

(*=======================================================*)
	6:	(* Konfigurationen der Achse *)
		IF fb_state_entry.E THEN
			fb_axis.st_eccoe_sdo.s_ec_slave_net_id := ST_EthercatDiag.s_ec_slave_net_id[2];
			fb_axis.st_eccoe_sdo.ui16_slave_addr := st_config_achse.ui16_ethercat_adr;
		END_IF

		(*-----------------------Weiterschaltbedingungen----------------------------*)
		fb_state_entry.i16_next_step := 7;

(*=======================================================*)
	7:	(* Spezifische NC-Achsparameter auslesen *)
		IF fb_state_entry.E THEN
			fb_axis.i16_nc_parameter_nummer := AxisMinSoftPosLimit;
			st_drive_cmd.enu_cmd := READ_NC_PARAMETER;
		END_IF

		(*-----------------------Weiterschaltbedingungen----------------------------*)
		IF st_drive_cmd.enu_cmd = NO_COMMAND THEN
			lr_MinSoftPosLimit := fb_axis.r_wert_nc_read_parameter;
			fb_state_entry.i16_next_step := 8;
		END_IF


(*=======================================================*)
	8:	(* Spezifische NC-Achsparameter auslesen *)
		IF fb_state_entry.E THEN
			fb_axis.i16_nc_parameter_nummer := AxisMaxSoftPosLimit;
			st_drive_cmd.enu_cmd := READ_NC_PARAMETER;
		END_IF

		(*-----------------------Weiterschaltbedingungen----------------------------*)
		IF st_drive_cmd.enu_cmd = NO_COMMAND THEN
			lr_MaxSoftPosLimit := fb_axis.r_wert_nc_read_parameter;
			fb_state_entry.i16_next_step := FEHLER; (*in Fehler gehen damit die Achsen resetet werden. Sonst steigen die Achsen bei einem TC Restart aus*)
		END_IF

(*=======================================================*)
	INIT:
		IF fb_state_entry.E THEN
			fb_ton_wz.IN := FALSE;
			fb_ton_uez.IN	:= FALSE;
			fb_ton_quitt.IN := FALSE;
			fb_ton_taktzeitmessung_wt_wechsel.IN := FALSE;
			fb_ton_taktzeitmessung_bestuecken.IN := FALSE;
			b_start_in:=FALSE;
			st_ctrl_in.b_start:=FALSE;
			st_ctrl_out.b_busy:=FALSE;
			st_ctrl_out.b_fehler := FALSE;
			st_ctrl_out.b_fertig := FALSE;
			st_ctrl_out.b_fertig_2 := FALSE;
			st_ctrl_out.b_bereit := FALSE;
			st_ctrl_out.b_gestoppt := FALSE;
			st_ctrl_out.b_prebereit := FALSE;
			axis_y_achse.st_ctrl.in.b_start := FALSE;
			i16_kollisionszaehler := 0;
			(* Reset Stoermeldungen *)
			st_sm.b_achse_nicht_auf_startpos := FALSE;
			st_sm.b_achsfehler := FALSE;
			st_sm.b_devicefehler := FALSE;
			st_sm.b_keine_verfahrfreigabe := FALSE;
			st_sm.b_ende_skalierungs_nocke := FALSE;
			st_sm.b_ende_camming_nocke := FALSE;
			st_sm.b_skalierung_noch_aktiv := FALSE;
			sm_positionsueberwachung := FALSE;
			sm_werkzeugreihenfolge_nicht_io := FALSE;
			sm_keine_bandfreigabe := FALSE;
			sm_tagnummer_ungueltig := FALSE;
			sm_typ_bestueckprogramm_falsch := FALSE;
			sm_keine_rafo_im_einzug:=FALSE;

			bm_rastnasen_1_fehlt := FALSE;
			bm_rastnasen_2_fehlt := FALSE;

			bm_kein_Pin_im_BB:= FALSE;

			axis_y_achse.st_ctrl.in.b_start := FALSE;
			axis_y_achse.st_ctrl.in.b_start_2 := FALSE;
			axis_virt_master.st_ctrl.in.b_start := FALSE;
			rasterfolienmontage.st_ctrl.in.b_start := FALSE;
			balluff_tag_reader.st_ctrl.in.b_start_lesen := FALSE;
			balluff_tag_reader.st_ctrl.in.b_start_schreiben := FALSE;

			b_kommt_von_init := TRUE;

			fb_axis.mc_buffermode_axis := MC_Aborting;

			fb_axis.lr_soll_geschwindigkeit := gst_datensatz.st_wkz.r_auto_z;

			st_geschwindigkeiten.lr_verzoegerung := lr_decceleration_normal;
		END_IF

		IF y_achse.NcToPlc.CoupleState > 0 THEN
			st_drive_cmd_y_achse.enu_cmd := CAM_OUT_SLAVE;
		END_IF

		(*-----------------------Weiterschaltbedingungen----------------------------*)
		IF st_ctrl_in.b_preinit THEN
			fb_state_entry.i16_next_step := 15;
		END_IF

(*=======================================================*)
	15:	(* Reglerfreigabe wegnehmen *)
		IF fb_state_entry.E THEN
			st_drive_cmd.enu_cmd := POWER_DISABLE;
		END_IF

		(*-----------------------Weiterschaltbedingungen----------------------------*)
		IF st_drive_cmd.enu_cmd = NO_COMMAND THEN
			fb_state_entry.i16_next_step := 20;
		END_IF

(*=======================================================*)
	20:	(* Überprüfe Nullpunktverschiebung des Absolutwertgebers auf Korrektheit *)
		IF fb_state_entry.E THEN
			fb_axis.i16_nc_parameter_nummer := AxisEncoderOffset;	(* vom Datentyp MC_AxisParameter *)
			st_drive_cmd.enu_cmd := READ_NC_PARAMETER;
		END_IF

		(*-----------------------Weiterschaltbedingungen----------------------------*)
		IF st_drive_cmd.enu_cmd = NO_COMMAND THEN
			IF fb_axis.r_wert_nc_read_parameter = gst_datensatz.st_md.st_md_z_achse.lr_nullpunktverschiebung THEN
				CASE gst_datensatz.st_md.i16_typ_zelle OF
					KEINE_ZELLE:
						;

					BESTUECKZELLE_1700, RASTERFOLIE:
						fb_state_entry.i16_next_step := 35;
	
					BESTUECKZELLE_1720:
						fb_state_entry.i16_next_step := 40;
				END_CASE
			ELSE
				fb_state_entry.i16_next_step := 25;	(* Nullpunktverschiebung schreiben *)
			END_IF
		END_IF

(*=======================================================*)
	25:	(* Nullpunktverschiebung hat sich geändert, deshalb erst Null reinschreiben, um keinen Additionsfehler zu machen, *)
		(* weil der Wert der Verschiebung beim Neustart komplett auf die Achse geschrieben wird *)
		IF fb_state_entry.E THEN
			fb_axis.i16_nc_parameter_nummer := AxisEncoderOffset;
			fb_axis.r_wert_nc_write_parameter := 0.0;
			st_drive_cmd.enu_cmd := WRITE_NC_PARAMETER;
		END_IF

		(*-----------------------Weiterschaltbedingungen----------------------------*)
		IF st_drive_cmd.enu_cmd = NO_COMMAND THEN
			fb_state_entry.i16_next_step := 30;
		END_IF

(*=======================================================*)
	30:	(* Aktuelle Nullpunktverschiebung des Absolutwertgebers an die Achse senden *)
		IF fb_state_entry.E THEN
			fb_axis.i16_nc_parameter_nummer := AxisEncoderOffset;
			fb_axis.r_wert_nc_write_parameter := gst_datensatz.st_md.st_md_z_achse.lr_nullpunktverschiebung;
			st_drive_cmd.enu_cmd := WRITE_NC_PARAMETER;
		END_IF

		(*-----------------------Weiterschaltbedingungen----------------------------*)
		IF st_drive_cmd.enu_cmd = NO_COMMAND THEN
			CASE gst_datensatz.st_md.i16_typ_zelle OF
				KEINE_ZELLE:
					;

				BESTUECKZELLE_1700, RASTERFOLIE:
					fb_state_entry.i16_next_step := 35;

